METHOD FB_init : BOOL
VAR_INPUT
	bInitRetains : BOOL; // if TRUE, the retain variables are initialized (warm start / cold start)
	bInCopyCode : BOOL;  // if TRUE, the instance afterwards gets moved into the copy code (online change)
END_VAR
eObjectType := E_BACnetObjType.ObjAnalogValue;
END_METHOD

END_FUNCTION_BLOCK

// POUs/Remote/Objects/Basic/[Base]/FB_BACnetRM_EventObject
FUNCTION_BLOCK FB_BACnetRM_EventObject EXTENDS FB_BACnetRM_Object
VAR_OUTPUT
	bEvent						: BOOL;												// Indicates an active event
END_VAR
VAR
	{region 'Event'}
		stStatusFlags			: ST_BA_StatusFlags;
	{endregion}
END_VAR

SUPER^();

bEvent := F_BA_IsDisturbed(stStatusFlags);

METHOD PROTECTED OnObjectStateChanged
SUPER^.OnObjectStateChanged();

SyncProperty(E_BACnetPropIdentifier.PropStatusFlags, SIZEOF(stStatusFlags), ADR(stStatusFlags), E_BA_SyncModeRM.eRead);
END_METHOD

PROPERTY StatusFlags : ST_BA_StatusFlags
GET
StatusFlags := stStatusFlags;
END_GET
END_PROPERTY

END_FUNCTION_BLOCK

// POUs/Remote/Objects/Basic/FB_BACnetRM_AV_Disp
{attribute 'enable_dynamic_creation'}
FUNCTION_BLOCK FB_BACnetRM_AV_Disp EXTENDS FB_BACnetRM_Object
VAR_INPUT CONSTANT PERSISTENT
	{region 'Fixed Parameters'}
		{attribute 'parameterCategory':='Config'}
		fReadIncrement : REAL;
	{endregion}
END_VAR
VAR_OUTPUT
	fPresVal 	: REAL;
END_VAR

SUPER^();

METHOD PROTECTED OnObjectStateChanged
SUPER^.OnObjectStateChanged();

SyncPropertyReal(E_BACnetPropIdentifier.PropPresentValue, SIZEOF(fPresVal), ADR(fPresVal), E_BA_SyncModeRM.eRead, fReadIncrement);
END_METHOD

METHOD FB_init : BOOL
VAR_INPUT
	bInitRetains : BOOL; // if TRUE, the retain variables are initialized (warm start / cold start)
	bInCopyCode : BOOL;  // if TRUE, the instance afterwards gets moved into the copy code (online change)
END_VAR
eObjectType := E_BACnetObjType.ObjAnalogValue;
END_METHOD

END_FUNCTION_BLOCK

// POUs/Remote/Objects/Basic/FB_BACnetRM_AV_Setp
{attribute 'enable_dynamic_creation'}
FUNCTION_BLOCK FB_BACnetRM_AV_Setp EXTENDS FB_BACnetRM_Object
VAR_INPUT CONSTANT PERSISTENT
	{region 'Fixed Parameters'}
		{attribute 'parameterCategory':='Config'}
		fReadIncrement : REAL; 
		{attribute 'parameterCategory':='Config'}
		fWriteIncrement : REAL; 
	{endregion}
END_VAR
VAR_INPUT CONSTANT
	{region 'Operational Parameters'}
		{attribute 'parameterCategory':='Value'}
		fValue : REAL;
	{endregion}
END_VAR
VAR_OUTPUT
	fPresVal 	: REAL;
END_VAR

SUPER^();

{attribute 'hide'}
METHOD OnCOV
VAR_INPUT
	ePropID		: E_BACnetPropIdentifier;
END_VAR
CASE (ePropID) OF
	E_BACnetPropIdentifier.PropPresentValue:
		fValue := fPresVal;
		
ELSE
	SUPER^.OnCOV(ePropID);
END_CASE
END_METHOD

METHOD PROTECTED OnObjectStateChanged
SUPER^.OnObjectStateChanged();

SyncPropertyReal(E_BACnetPropIdentifier.PropPresentValue, SIZEOF(fPresVal), ADR(fPresVal), E_BA_SyncModeRM.eRead, fReadIncrement);

SyncPropertyReal(E_BACnetPropIdentifier.PropPresentValue, SIZEOF(fValue), ADR(fValue), E_BA_SyncModeRM.eWrite, fWriteIncrement);
END_METHOD

METHOD FB_init : BOOL
VAR_INPUT
	bInitRetains : BOOL; // if TRUE, the retain variables are initialized (warm start / cold start)
	bInCopyCode : BOOL;  // if TRUE, the instance afterwards gets moved into the copy code (online change)
END_VAR
eObjectType := E_BACnetObjType.ObjAnalogValue;
END_METHOD

END_FUNCTION_BLOCK

// POUs/Remote/Objects/Basic/FB_BACnetRM_AI
{attribute 'enable_dynamic_creation'}
FUNCTION_BLOCK FB_BACnetRM_AI EXTENDS FB_BACnetRM_EventObject
VAR_INPUT CONSTANT PERSISTENT
	{region 'Fixed Parameters'}
		{attribute 'parameterCategory':='Config'}
		fReadIncrement : REAL; 
	{endregion}
END_VAR
VAR_OUTPUT
	fPresVal 	: REAL;
END_VAR

SUPER^();

METHOD PROTECTED OnObjectStateChanged
SUPER^.OnObjectStateChanged();

SyncPropertyReal(E_BACnetPropIdentifier.PropPresentValue, SIZEOF(fPresVal), ADR(fPresVal), E_BA_SyncModeRM.eRead, fReadIncrement);
END_METHOD

METHOD FB_init : BOOL
VAR_INPUT
	bInitRetains : BOOL; // if TRUE, the retain variables are initialized (warm start / cold start)
	bInCopyCode : BOOL;  // if TRUE, the instance afterwards gets moved into the copy code (online change)
END_VAR
eObjectType := E_BACnetObjType.ObjAnalogInput;
END_METHOD

END_FUNCTION_BLOCK

// POUs/Remote/Objects/Basic/FB_BACnetRM_AO
{attribute 'enable_dynamic_creation'}
FUNCTION_BLOCK FB_BACnetRM_AO EXTENDS FB_BACnetRM_EventObject
VAR_INPUT
	bEnWrite	 	: BOOL;
	fVal 			: REAL;
	bNullVal 		: BOOL;
END_VAR
VAR_INPUT CONSTANT PERSISTENT
	{region 'Fixed Parameters'}
		{attribute 'parameterCategory':='Config'}
		fReadIncrement : REAL; 
		{attribute 'parameterCategory':='Config'}
		fWriteIncrement : REAL; 
			 
		{attribute 'parameterCategory':='Value'}
		ePriority : E_BACnet_Priority := BACnet_Param.eRemotePrio_Default;
	{endregion}
END_VAR
VAR_OUTPUT
	fPresVal 	: REAL;
END_VAR

SUPER^();

METHOD PROTECTED OnObjectStateChanged
SUPER^.OnObjectStateChanged();

SyncPropertyReal(E_BACnetPropIdentifier.PropPresentValue, SIZEOF(fPresVal), ADR(fPresVal), E_BA_SyncModeRM.eRead, fReadIncrement);

SyncPropertyPrioReal(E_BACnetPropIdentifier.PropPresentValue, SIZEOF(fVal), ADR(fVal), ADR(bEnWrite), ADR(bNullVal), ePriority, E_BA_SyncModeRM.eWrite, fWriteIncrement);
END_METHOD

METHOD FB_init : BOOL
VAR_INPUT
	bInitRetains : BOOL; // if TRUE, the retain variables are initialized (warm start / cold start)
	bInCopyCode : BOOL;  // if TRUE, the instance afterwards gets moved into the copy code (online change)
END_VAR
eObjectType := E_BACnetObjType.ObjAnalogOutput;
END_METHOD

END_FUNCTION_BLOCK

// POUs/Remote/Objects/Basic/FB_BACnetRM_BV
{attribute 'enable_dynamic_creation'}
FUNCTION_BLOCK FB_BACnetRM_BV EXTENDS FB_BACnetRM_EventObject
VAR_INPUT
	bEnWrite 		: BOOL;
	bVal 			: BOOL;
	bNullVal 		: BOOL;
END_VAR
VAR_INPUT CONSTANT PERSISTENT
	{region 'Fixed Parameters'}
		{attribute 'parameterCategory':='Value'}
		ePriority : E_BACnet_Priority := BACnet_Param.eRemotePrio_Default;
	{endregion}
END_VAR
VAR_OUTPUT
	bPresVal 	: BOOL;
END_VAR

SUPER^();

METHOD PROTECTED OnObjectStateChanged
SUPER^.OnObjectStateChanged();

SyncProperty(E_BACnetPropIdentifier.PropPresentValue, SIZEOF(bPresVal), ADR(bPresVal), E_BA_SyncModeRM.eRead);

SyncPropertyPrio(E_BACnetPropIdentifier.PropPresentValue, SIZEOF(bVal), ADR(bVal), ADR(bEnWrite), ADR(bNullVal), ePriority, E_BA_SyncModeRM.eWrite);
END_METHOD

METHOD FB_init : BOOL
VAR_INPUT
	bInitRetains : BOOL; // if TRUE, the retain variables are initialized (warm start / cold start)
	bInCopyCode : BOOL;  // if TRUE, the instance afterwards gets moved into the copy code (online change)
END_VAR
eObjectType := E_BACnetObjType.ObjBinaryValue;
END_METHOD

END_FUNCTION_BLOCK

// POUs/Remote/Objects/Basic/FB_BACnetRM_BV_Disp
{attribute 'enable_dynamic_creation'}
FUNCTION_BLOCK FB_BACnetRM_BV_Disp EXTENDS FB_BACnetRM_Object
VAR_OUTPUT
	bPresVal	: BOOL;
END_VAR

SUPER^();

METHOD PROTECTED OnObjectStateChanged
SUPER^.OnObjectStateChanged();

SyncProperty(E_BACnetPropIdentifier.PropPresentValue, SIZEOF(bPresVal), ADR(bPresVal), E_BA_SyncModeRM.eRead);
END_METHOD

METHOD FB_init : BOOL
VAR_INPUT
	bInitRetains : BOOL; // if TRUE, the retain variables are initialized (warm start / cold start)
	bInCopyCode : BOOL;  // if TRUE, the instance afterwards gets moved into the copy code (online change)
END_VAR
eObjectType := E_BACnetObjType.ObjBinaryValue;
END_METHOD

END_FUNCTION_BLOCK

// POUs/Remote/Objects/Basic/FB_BACnetRM_BV_Setp
{attribute 'enable_dynamic_creation'}
FUNCTION_BLOCK FB_BACnetRM_BV_Setp EXTENDS FB_BACnetRM_Object
VAR_INPUT CONSTANT
	{region 'Operational Parameters'}
		{attribute 'parameterCategory':='Value'}
		bValue : BOOL;
	{endregion}
END_VAR
VAR_OUTPUT
	bPresVal	: BOOL;
END_VAR

SUPER^();

{attribute 'hide'}
METHOD OnCOV
VAR_INPUT
	ePropID		: E_BACnetPropIdentifier;
END_VAR
CASE (ePropID) OF
	E_BACnetPropIdentifier.PropPresentValue:
		bValue := bPresVal;
		
ELSE
	SUPER^.OnCOV(ePropID);
END_CASE
END_METHOD

METHOD PROTECTED OnObjectStateChanged
SUPER^.OnObjectStateChanged();

SyncProperty(E_BACnetPropIdentifier.PropPresentValue, SIZEOF(bPresVal), ADR(bPresVal), E_BA_SyncModeRM.eRead);

SyncProperty(E_BACnetPropIdentifier.PropPresentValue, SIZEOF(bValue), ADR(bValue), E_BA_SyncModeRM.eWrite);
END_METHOD

METHOD FB_init : BOOL
VAR_INPUT
	bInitRetains : BOOL; // if TRUE, the retain variables are initialized (warm start / cold start)
	bInCopyCode : BOOL;  // if TRUE, the instance afterwards gets moved into the copy code (online change)
END_VAR
eObjectType := E_BACnetObjType.ObjBinaryValue;
END_METHOD

END_FUNCTION_BLOCK

// POUs/Remote/Objects/Basic/FB_BACnetRM_BI
{attribute 'enable_dynamic_creation'}
FUNCTION_BLOCK FB_BACnetRM_BI EXTENDS FB_BACnetRM_EventObject
VAR_OUTPUT
	bPresVal 	: BOOL;
END_VAR

SUPER^();

METHOD PROTECTED OnObjectStateChanged
SUPER^.OnObjectStateChanged();

SyncProperty(E_BACnetPropIdentifier.PropPresentValue, SIZEOF(bPresVal), ADR(bPresVal), E_BA_SyncModeRM.eRead);
END_METHOD

METHOD FB_init : BOOL
VAR_INPUT
	bInitRetains : BOOL; // if TRUE, the retain variables are initialized (warm start / cold start)
	bInCopyCode : BOOL;  // if TRUE, the instance afterwards gets moved into the copy code (online change)
END_VAR
eObjectType := E_BACnetObjType.ObjBinaryInput;
END_METHOD

END_FUNCTION_BLOCK

// POUs/Remote/Objects/Basic/FB_BACnetRM_BO
{attribute 'enable_dynamic_creation'}
FUNCTION_BLOCK FB_BACnetRM_BO EXTENDS FB_BACnetRM_EventObject
VAR_INPUT
	bEnWrite 		: BOOL;
	bVal 			: BOOL;
	bNullVal 		: BOOL;	
END_VAR
VAR_INPUT CONSTANT PERSISTENT
	{region 'Fixed Parameters'}
		{attribute 'parameterCategory':='Value'}
		ePriority : E_BACnet_Priority := BACnet_Param.eRemotePrio_Default;
	{endregion}
END_VAR
VAR_OUTPUT
	bPresVal 	: BOOL;
END_VAR

SUPER^();

METHOD PROTECTED OnObjectStateChanged
SUPER^.OnObjectStateChanged();

SyncProperty(E_BACnetPropIdentifier.PropPresentValue, SIZEOF(bPresVal), ADR(bPresVal), E_BA_SyncModeRM.eRead);

SyncPropertyPrio(E_BACnetPropIdentifier.PropPresentValue, SIZEOF(bVal), ADR(bVal), ADR(bEnWrite), ADR(bNullVal), ePriority, E_BA_SyncModeRM.eWrite);
END_METHOD

METHOD FB_init : BOOL
VAR_INPUT
	bInitRetains : BOOL; // if TRUE, the retain variables are initialized (warm start / cold start)
	bInCopyCode : BOOL;  // if TRUE, the instance afterwards gets moved into the copy code (online change)
END_VAR
eObjectType := E_BACnetObjType.ObjBinaryOutput;
END_METHOD

END_FUNCTION_BLOCK

// POUs/Remote/Objects/Basic/FB_BACnetRM_MV
{attribute 'enable_dynamic_creation'}
FUNCTION_BLOCK FB_BACnetRM_MV EXTENDS FB_BACnetRM_EventObject
VAR_INPUT
	bEnWrite 		: BOOL;
	nVal 			: UDINT;
	bNullVal 		: BOOL;	
END_VAR
VAR_INPUT CONSTANT PERSISTENT
	{region 'Fixed Parameters'}
		{attribute 'parameterCategory':='Value'}
		ePriority : E_BACnet_Priority := BACnet_Param.eRemotePrio_Default;
	{endregion}
END_VAR
VAR_OUTPUT
	nPresVal 	: UDINT;
END_VAR

SUPER^();

METHOD PROTECTED OnObjectStateChanged
SUPER^.OnObjectStateChanged();

SyncProperty(E_BACnetPropIdentifier.PropPresentValue, SIZEOF(nPresVal), ADR(nPresVal), E_BA_SyncModeRM.eRead);

SyncPropertyPrio(E_BACnetPropIdentifier.PropPresentValue, SIZEOF(nVal), ADR(nVal), ADR(bEnWrite), ADR(bNullVal), ePriority, E_BA_SyncModeRM.eWrite);
END_METHOD

METHOD FB_init : BOOL
VAR_INPUT
	bInitRetains : BOOL; // if TRUE, the retain variables are initialized (warm start / cold start)
	bInCopyCode : BOOL;  // if TRUE, the instance afterwards gets moved into the copy code (online change)
END_VAR
eObjectType := E_BACnetObjType.ObjMultistateValue;
END_METHOD

END_FUNCTION_BLOCK

// POUs/Remote/Objects/Basic/FB_BACnetRM_MV_Disp
{attribute 'enable_dynamic_creation'}
FUNCTION_BLOCK FB_BACnetRM_MV_Disp EXTENDS FB_BACnetRM_Object
VAR_OUTPUT
	nPresVal		: UDINT		:= 1;
END_VAR

SUPER^();

METHOD PROTECTED OnObjectStateChanged
SUPER^.OnObjectStateChanged();

SyncProperty(E_BACnetPropIdentifier.PropPresentValue, SIZEOF(nPresVal), ADR(nPresVal), E_BA_SyncModeRM.eRead);
END_METHOD

METHOD FB_init : BOOL
VAR_INPUT
	bInitRetains : BOOL; // if TRUE, the retain variables are initialized (warm start / cold start)
	bInCopyCode : BOOL;  // if TRUE, the instance afterwards gets moved into the copy code (online change)
END_VAR
eObjectType := E_BACnetObjType.ObjMultistateValue;
END_METHOD

END_FUNCTION_BLOCK

// POUs/Remote/Objects/Basic/FB_BACnetRM_MV_Setp
{attribute 'enable_dynamic_creation'}
FUNCTION_BLOCK FB_BACnetRM_MV_Setp EXTENDS FB_BACnetRM_Object
VAR_INPUT CONSTANT
	{region 'Operational Parameters'}
		{attribute 'parameterCategory':='Value'}
		nValue : UDINT;
	{endregion}
END_VAR
VAR_OUTPUT
	nPresVal		: UDINT		:= 1;
END_VAR

SUPER^();

{attribute 'hide'}
METHOD OnCOV
VAR_INPUT
	ePropID		: E_BACnetPropIdentifier;
END_VAR
CASE (ePropID) OF
	E_BACnetPropIdentifier.PropPresentValue:
		nValue := nPresVal;
		
ELSE
	SUPER^.OnCOV(ePropID);
END_CASE
END_METHOD

METHOD PROTECTED OnObjectStateChanged
SUPER^.OnObjectStateChanged();

SyncProperty(E_BACnetPropIdentifier.PropPresentValue, SIZEOF(nPresVal), ADR(nPresVal), E_BA_SyncModeRM.eRead);

SyncProperty(E_BACnetPropIdentifier.PropPresentValue, SIZEOF(nValue), ADR(nValue), E_BA_SyncModeRM.eWrite);
END_METHOD

METHOD FB_init : BOOL
VAR_INPUT
	bInitRetains : BOOL; // if TRUE, the retain variables are initialized (warm start / cold start)
	bInCopyCode : BOOL;  // if TRUE, the instance afterwards gets moved into the copy code (online change)
END_VAR
eObjectType := E_BACnetObjType.ObjMultistateValue;
END_METHOD

END_FUNCTION_BLOCK

// POUs/Remote/Objects/Basic/FB_BACnetRM_MI
{attribute 'enable_dynamic_creation'}
FUNCTION_BLOCK FB_BACnetRM_MI EXTENDS FB_BACnetRM_EventObject
VAR_OUTPUT
	nPresVal 	: UDINT;
END_VAR

SUPER^();

METHOD PROTECTED OnObjectStateChanged
SUPER^.OnObjectStateChanged();

SyncProperty(E_BACnetPropIdentifier.PropPresentValue, SIZEOF(nPresVal), ADR(nPresVal), E_BA_SyncModeRM.eRead);
END_METHOD

METHOD FB_init : BOOL
VAR_INPUT
	bInitRetains : BOOL; // if TRUE, the retain variables are initialized (warm start / cold start)
	bInCopyCode : BOOL;  // if TRUE, the instance afterwards gets moved into the copy code (online change)
END_VAR
eObjectType := E_BACnetObjType.ObjMultistateInput;
END_METHOD

END_FUNCTION_BLOCK

// POUs/Remote/Objects/Basic/FB_BACnetRM_MO
{attribute 'enable_dynamic_creation'}
FUNCTION_BLOCK FB_BACnetRM_MO EXTENDS FB_BACnetRM_EventObject
VAR_INPUT
	bEnWrite 		: BOOL;
	nVal 			: UDINT;
	bNullVal 		: BOOL;
END_VAR
VAR_INPUT CONSTANT PERSISTENT
	{region 'Fixed Parameters'}
		{attribute 'parameterCategory':='Value'}
		ePriority : E_BACnet_Priority := BACnet_Param.eRemotePrio_Default;
	{endregion}
END_VAR
VAR_OUTPUT
	nPresVal 	: UDINT;
END_VAR

SUPER^();

METHOD PROTECTED OnObjectStateChanged
SUPER^.OnObjectStateChanged();

SyncProperty(E_BACnetPropIdentifier.PropPresentValue, SIZEOF(nPresVal), ADR(nPresVal), E_BA_SyncModeRM.eRead);

SyncPropertyPrio(E_BACnetPropIdentifier.PropPresentValue, SIZEOF(nVal), ADR(nVal), ADR(bEnWrite), ADR(bNullVal), ePriority, E_BA_SyncModeRM.eWrite);
END_METHOD

METHOD FB_init : BOOL
VAR_INPUT
	bInitRetains : BOOL; // if TRUE, the retain variables are initialized (warm start / cold start)
	bInCopyCode : BOOL;  // if TRUE, the instance afterwards gets moved into the copy code (online change)
END_VAR
eObjectType := E_BACnetObjType.ObjMultistateOutput;
END_METHOD

END_FUNCTION_BLOCK

// POUs/Remote/Objects/Basic/FB_BACnetRM_TLog
{attribute 'enable_dynamic_creation'}
FUNCTION_BLOCK FB_BACnetRM_TLog EXTENDS FB_BACnetRM_BaseTLog
VAR_OUTPUT
	nRecCnt 	: UDINT;
	nTotRecCnt	: UDINT;
END_VAR

SUPER^();

METHOD PROTECTED OnObjectStateChanged
SUPER^.OnObjectStateChanged();

SyncProperty(E_BACnetPropIdentifier.PropRecordCount, SIZEOF(nRecCnt), ADR(nRecCnt), E_BA_SyncModeRM.eRead);
SyncProperty(E_BACnetPropIdentifier.PropTotalRecordCount, SIZEOF(nTotRecCnt), ADR(nTotRecCnt), E_BA_SyncModeRM.eRead);
END_METHOD

METHOD FB_init : BOOL
VAR_INPUT
	bInitRetains : BOOL; // if TRUE, the retain variables are initialized (warm start / cold start)
	bInCopyCode : BOOL;  // if TRUE, the instance afterwards gets moved into the copy code (online change)
END_VAR
eObjectType := E_BACnetObjType.ObjTrendLog;
END_METHOD

END_FUNCTION_BLOCK

// POUs/Remote/Objects/Basic/[Base]/FB_BACnetRM_BaseTLog
FUNCTION_BLOCK FB_BACnetRM_BaseTLog EXTENDS FB_BACnetRM_EventObject
VAR_OUTPUT
	nRecordCount				: UDINT;
	nTotalRecordCount			: UDINT;
END_VAR

SUPER^();

METHOD PROTECTED OnObjectStateChanged
SUPER^.OnObjectStateChanged();

SyncProperty(E_BACnetPropIdentifier.PropRecordCount, SIZEOF(nRecordCount), ADR(nRecordCount), E_BA_SyncModeRM.eRead);
SyncProperty(E_BACnetPropIdentifier.PropTotalRecordCount, SIZEOF(nTotalRecordCount), ADR(nTotalRecordCount), E_BA_SyncModeRM.eRead);
END_METHOD

END_FUNCTION_BLOCK

// POUs/Remote/Objects/Basic/FB_BACnetRM_TLM
{attribute 'enable_dynamic_creation'}
FUNCTION_BLOCK FB_BACnetRM_TLM EXTENDS FB_BACnetRM_BaseTLog
VAR_OUTPUT
	nRecCnt 	: UDINT;
	nTotRecCnt	: UDINT;
END_VAR

SUPER^();

METHOD PROTECTED OnObjectStateChanged
SUPER^.OnObjectStateChanged();

SyncProperty(E_BACnetPropIdentifier.PropRecordCount, SIZEOF(nRecCnt), ADR(nRecCnt), E_BA_SyncModeRM.eRead);
SyncProperty(E_BACnetPropIdentifier.PropTotalRecordCount, SIZEOF(nTotRecCnt), ADR(nTotRecCnt), E_BA_SyncModeRM.eRead);
END_METHOD

METHOD FB_init : BOOL
VAR_INPUT
	bInitRetains : BOOL; // if TRUE, the retain variables are initialized (warm start / cold start)
	bInCopyCode : BOOL;  // if TRUE, the instance afterwards gets moved into the copy code (online change)
END_VAR
eObjectType := E_BACnetObjType.ObjTrendLogMultiple;
END_METHOD

END_FUNCTION_BLOCK

// POUs/Remote/Objects/Basic/FB_BACnetRM_Cal
{attribute 'enable_dynamic_creation'}
FUNCTION_BLOCK FB_BACnetRM_Cal EXTENDS FB_BACnetRM_Object
VAR_OUTPUT
	bPresVal 	: BOOL;
END_VAR

SUPER^();

METHOD PROTECTED OnObjectStateChanged
SUPER^.OnObjectStateChanged();

SyncProperty(E_BACnetPropIdentifier.PropPresentValue, SIZEOF(bPresVal), ADR(bPresVal), E_BA_SyncModeRM.eRead);
END_METHOD

METHOD FB_init : BOOL
VAR_INPUT
	bInitRetains : BOOL; // if TRUE, the retain variables are initialized (warm start / cold start)
	bInCopyCode : BOOL;  // if TRUE, the instance afterwards gets moved into the copy code (online change)
END_VAR
eObjectType := E_BACnetObjType.ObjCalendar;
END_METHOD

END_FUNCTION_BLOCK

// POUs/Remote/Objects/Basic/FB_BACnetRM_SchedA
{attribute 'enable_dynamic_creation'}
FUNCTION_BLOCK FB_BACnetRM_SchedA EXTENDS FB_BACnetRM_Object
VAR_OUTPUT
	fPresVal 	: REAL;
END_VAR

SUPER^();

METHOD PROTECTED OnObjectStateChanged
SUPER^.OnObjectStateChanged();

SyncProperty(E_BACnetPropIdentifier.PropPresentValue, SIZEOF(fPresVal), ADR(fPresVal), E_BA_SyncModeRM.eRead);
END_METHOD

METHOD FB_init : BOOL
VAR_INPUT
	bInitRetains : BOOL; // if TRUE, the retain variables are initialized (warm start / cold start)
	bInCopyCode : BOOL;  // if TRUE, the instance afterwards gets moved into the copy code (online change)
END_VAR
eObjectType := E_BACnetObjType.ObjSchedule;
END_METHOD

END_FUNCTION_BLOCK

// POUs/Remote/Objects/Basic/FB_BACnetRM_SchedB
{attribute 'enable_dynamic_creation'}
FUNCTION_BLOCK FB_BACnetRM_SchedB EXTENDS FB_BACnetRM_Object
VAR_OUTPUT
	bPresVal 	: BOOL;
END_VAR

SUPER^();

METHOD PROTECTED OnObjectStateChanged
SUPER^.OnObjectStateChanged();

SyncProperty(E_BACnetPropIdentifier.PropPresentValue, SIZEOF(bPresVal), ADR(bPresVal), E_BA_SyncModeRM.eRead);
END_METHOD

METHOD FB_init : BOOL
VAR_INPUT
	bInitRetains : BOOL; // if TRUE, the retain variables are initialized (warm start / cold start)
	bInCopyCode : BOOL;  // if TRUE, the instance afterwards gets moved into the copy code (online change)
END_VAR
eObjectType := E_BACnetObjType.ObjSchedule;
END_METHOD

END_FUNCTION_BLOCK

// POUs/Remote/Objects/Basic/FB_BACnetRM_SchedM
{attribute 'enable_dynamic_creation'}
FUNCTION_BLOCK FB_BACnetRM_SchedM EXTENDS FB_BACnetRM_Object
VAR_OUTPUT
	nPresVal 	: UDINT;
END_VAR

SUPER^();

METHOD PROTECTED OnObjectStateChanged
SUPER^.OnObjectStateChanged();

SyncProperty(E_BACnetPropIdentifier.PropPresentValue, SIZEOF(nPresVal), ADR(nPresVal), E_BA_SyncModeRM.eRead);
END_METHOD

METHOD FB_init : BOOL
VAR_INPUT
	bInitRetains : BOOL; // if TRUE, the retain variables are initialized (warm start / cold start)
	bInCopyCode : BOOL;  // if TRUE, the instance afterwards gets moved into the copy code (online change)
END_VAR
eObjectType := E_BACnetObjType.ObjSchedule;
END_METHOD

END_FUNCTION_BLOCK

// POUs/Remote/Objects/Basic/FB_BACnetRM_Loop
{attribute 'enable_dynamic_creation'}
FUNCTION_BLOCK FB_BACnetRM_Loop EXTENDS FB_BACnetRM_EventObject
VAR_OUTPUT
	fPresVal			: REAL;
	fSetpoint			: REAL;
	fCtrlVar			: REAL;
END_VAR

SUPER^();

METHOD PROTECTED OnObjectStateChanged
SUPER^.OnObjectStateChanged();

SyncProperty(E_BACnetPropIdentifier.PropPresentValue, SIZEOF(fPresVal), ADR(fPresVal), E_BA_SyncModeRM.eRead);
SyncProperty(E_BACnetPropIdentifier.PropSetpoint, SIZEOF(fSetpoint), ADR(fSetpoint), E_BA_SyncModeRM.eRead);
SyncProperty(E_BACnetPropIdentifier.PropControlledVariableValue, SIZEOF(fCtrlVar), ADR(fCtrlVar), E_BA_SyncModeRM.eRead);
END_METHOD

METHOD FB_init : BOOL
VAR_INPUT
	bInitRetains : BOOL; // if TRUE, the retain variables are initialized (warm start / cold start)
	bInCopyCode : BOOL;  // if TRUE, the instance afterwards gets moved into the copy code (online change)
END_VAR
eObjectType := E_BACnetObjType.ObjLoop;
END_METHOD

END_FUNCTION_BLOCK

// POUs/Remote/Objects/Convenience/FB_BACnetRM_CnvLoop
{attribute 'enable_dynamic_creation'}
FUNCTION_BLOCK FB_BACnetRM_CnvLoop EXTENDS FB_BACnetRM_Loop
VAR_INPUT CONSTANT PERSISTENT
	{region 'Variable Parameters'}
		{attribute 'parameterCategory':='Config'}
		fProportionalConstant : REAL;
		{attribute 'parameterCategory':='Config'}
		eProportionalConstantUnit : E_BA_Unit;
		{attribute 'parameterCategory':='Config'}
		fIntegralConstant : REAL;
		{attribute 'parameterCategory':='Config'}
		eIntegralConstantUnit : E_BA_Unit;
		{attribute 'parameterCategory':='Config'}
		fDerivativeConstant : REAL;
		{attribute 'parameterCategory':='Config'}
		eDerivativeConstantUnit : E_BA_Unit;
	{endregion}
END_VAR

SUPER^();

METHOD PROTECTED OnObjectStateChanged
SUPER^.OnObjectStateChanged();

SyncProperty(E_BACnetPropIdentifier.PropProportionalConstant, SIZEOF(fProportionalConstant), ADR(fProportionalConstant), E_BA_SyncModeRM.eRead);
SyncProperty(E_BACnetPropIdentifier.PropProportionalConstantUnits, SIZEOF(eProportionalConstantUnit), ADR(eProportionalConstantUnit), E_BA_SyncModeRM.eRead);
SyncProperty(E_BACnetPropIdentifier.PropIntegralConstant, SIZEOF(fIntegralConstant), ADR(fIntegralConstant), E_BA_SyncModeRM.eRead);
SyncProperty(E_BACnetPropIdentifier.PropIntegralConstantUnits, SIZEOF(eIntegralConstantUnit), ADR(eIntegralConstantUnit), E_BA_SyncModeRM.eRead);
SyncProperty(E_BACnetPropIdentifier.PropDerivativeConstant, SIZEOF(fDerivativeConstant), ADR(fDerivativeConstant), E_BA_SyncModeRM.eRead);
SyncProperty(E_BACnetPropIdentifier.PropDerivativeConstantUnits, SIZEOF(eDerivativeConstantUnit), ADR(eDerivativeConstantUnit), E_BA_SyncModeRM.eRead);
END_METHOD

END_FUNCTION_BLOCK

// POUs/Remote/Objects/Basic/FB_BACnetRM_File
{attribute 'enable_dynamic_creation'}
FUNCTION_BLOCK FB_BACnetRM_File EXTENDS FB_BACnetRM_Object
VAR_OUTPUT
	nFileSize		: UDINT;
END_VAR

SUPER^();

METHOD PROTECTED OnObjectStateChanged
SUPER^.OnObjectStateChanged();

SyncProperty(E_BACnetPropIdentifier.PropFileSize, SIZEOF(nFileSize), ADR(nFileSize), E_BA_SyncModeRM.eRead);
END_METHOD

METHOD FB_init : BOOL
VAR_INPUT
	bInitRetains : BOOL; // if TRUE, the retain variables are initialized (warm start / cold start)
	bInCopyCode : BOOL;  // if TRUE, the instance afterwards gets moved into the copy code (online change)
END_VAR
eObjectType := E_BACnetObjType.ObjFile;
END_METHOD

END_FUNCTION_BLOCK

// POUs/Remote/Objects/Basic/FB_BACnetRM_NC
{attribute 'enable_dynamic_creation'}
FUNCTION_BLOCK FB_BACnetRM_NC EXTENDS FB_BACnetRM_Object

SUPER^();

METHOD FB_init : BOOL
VAR_INPUT
	bInitRetains : BOOL; // if TRUE, the retain variables are initialized (warm start / cold start)
	bInCopyCode : BOOL;  // if TRUE, the instance afterwards gets moved into the copy code (online change)
END_VAR
eObjectType := E_BACnetObjType.ObjNotificationClass;
END_METHOD

END_FUNCTION_BLOCK

// POUs/Remote/Objects/Basic/FB_BACnetRM_Acc
{attribute 'enable_dynamic_creation'}
FUNCTION_BLOCK FB_BACnetRM_Acc EXTENDS FB_BACnetRM_EventObject
VAR_OUTPUT
	nPresVal			: UDINT;
END_VAR

SUPER^();

METHOD PROTECTED OnObjectStateChanged
SUPER^.OnObjectStateChanged();

SyncProperty(E_BACnetPropIdentifier.PropPresentValue, SIZEOF(nPresVal), ADR(nPresVal), E_BA_SyncModeRM.eRead);
END_METHOD

METHOD FB_init : BOOL
VAR_INPUT
	bInitRetains : BOOL; // if TRUE, the retain variables are initialized (warm start / cold start)
	bInCopyCode : BOOL;  // if TRUE, the instance afterwards gets moved into the copy code (online change)
END_VAR
eObjectType := E_BACnetObjType.ObjAccumulator;
END_METHOD

END_FUNCTION_BLOCK

// POUs/Remote/Objects/Basic/FB_BACnetRM_PC
{attribute 'enable_dynamic_creation'}
FUNCTION_BLOCK FB_BACnetRM_PC EXTENDS FB_BACnetRM_EventObject
VAR_OUTPUT
	fPresVal			: REAL;
END_VAR

SUPER^();

METHOD PROTECTED OnObjectStateChanged
SUPER^.OnObjectStateChanged();

SyncProperty(E_BACnetPropIdentifier.PropPresentValue, SIZEOF(fPresVal), ADR(fPresVal), E_BA_SyncModeRM.eRead);
END_METHOD

METHOD FB_init : BOOL
VAR_INPUT
	bInitRetains : BOOL; // if TRUE, the retain variables are initialized (warm start / cold start)
	bInCopyCode : BOOL;  // if TRUE, the instance afterwards gets moved into the copy code (online change)
END_VAR
eObjectType := E_BACnetObjType.ObjPulseConverter;
END_METHOD

END_FUNCTION_BLOCK

// POUs/Remote/Objects/Basic/FB_BACnetRM_Prog
{attribute 'enable_dynamic_creation'}
FUNCTION_BLOCK FB_BACnetRM_Prog EXTENDS FB_BACnetRM_EventObject
VAR_OUTPUT
	eState			: E_BACnet_ProgramState;
END_VAR

SUPER^();

METHOD PROTECTED OnObjectStateChanged
SUPER^.OnObjectStateChanged();

SyncProperty(E_BACnetPropIdentifier.PropProgramState, SIZEOF(eState), ADR(eState), E_BA_SyncModeRM.eRead);
END_METHOD

METHOD FB_init : BOOL
VAR_INPUT
	bInitRetains : BOOL; // if TRUE, the retain variables are initialized (warm start / cold start)
	bInCopyCode : BOOL;  // if TRUE, the instance afterwards gets moved into the copy code (online change)
END_VAR
eObjectType := E_BACnetObjType.ObjProg;
END_METHOD

END_FUNCTION_BLOCK

// POUs/Remote/Objects/Basic/FB_BACnetRM_Avg
{attribute 'enable_dynamic_creation'}
FUNCTION_BLOCK FB_BACnetRM_Avg EXTENDS FB_BACnetRM_Object
VAR_OUTPUT
	fAvgVal			: REAL;
	fMinVal			: REAL;
	fMaxVal			: REAL;
END_VAR

SUPER^();

METHOD PROTECTED OnObjectStateChanged
VAR
	nPresentValue: INT;
END_VAR
SUPER^.OnObjectStateChanged();

SyncProperty(E_BACnetPropIdentifier.PropAverageValue, SIZEOF(fAvgVal), ADR(fAvgVal), E_BA_SyncModeRM.eRead);
SyncProperty(E_BACnetPropIdentifier.PropMinimumValue, SIZEOF(fMinVal), ADR(fMinVal), E_BA_SyncModeRM.eRead);
SyncProperty(E_BACnetPropIdentifier.PropMaximumValue, SIZEOF(fMaxVal), ADR(fMaxVal), E_BA_SyncModeRM.eRead);
END_METHOD

METHOD FB_init : BOOL
VAR_INPUT
	bInitRetains : BOOL; // if TRUE, the retain variables are initialized (warm start / cold start)
	bInCopyCode : BOOL;  // if TRUE, the instance afterwards gets moved into the copy code (online change)
END_VAR
eObjectType := E_BACnetObjType.ObjAveraging;
END_METHOD

END_FUNCTION_BLOCK

// POUs/Remote/Objects/Basic/FB_BACnetRM_Cmd
{attribute 'enable_dynamic_creation'}
FUNCTION_BLOCK FB_BACnetRM_Cmd EXTENDS FB_BACnetRM_Object
VAR_OUTPUT
	nPresVal			: UDINT;
	bAllWritesOk		: BOOL; (* all actions in selected action list are written *)
	bInProcess			: BOOL; (* object is busy *)
END_VAR

SUPER^();

METHOD PROTECTED OnObjectStateChanged
SUPER^.OnObjectStateChanged();

SyncProperty(E_BACnetPropIdentifier.PropPresentValue, SIZEOF(nPresVal), ADR(nPresVal), E_BA_SyncModeRM.eRead);
SyncProperty(E_BACnetPropIdentifier.PropAllWritesSuccessful, SIZEOF(bAllWritesOk), ADR(bAllWritesOk), E_BA_SyncModeRM.eRead);
SyncProperty(E_BACnetPropIdentifier.PropInProcess, SIZEOF(bInProcess), ADR(bInProcess), E_BA_SyncModeRM.eRead);
END_METHOD

METHOD FB_init : BOOL
VAR_INPUT
	bInitRetains : BOOL; // if TRUE, the retain variables are initialized (warm start / cold start)
	bInCopyCode : BOOL;  // if TRUE, the instance afterwards gets moved into the copy code (online change)
END_VAR
eObjectType := E_BACnetObjType.ObjCommand;
END_METHOD

END_FUNCTION_BLOCK

// POUs/Remote/Objects/Basic/FB_BACnetRM_Device
{attribute 'enable_dynamic_creation'}
FUNCTION_BLOCK FB_BACnetRM_Device EXTENDS FB_BACnetRM_Object
VAR_OUTPUT
	bOperational		: BOOL;
END_VAR

IF (NOT bReady) THEN
	IF (nObjectInstance = BACnet_Globals.nBACnetInstId_Auto) THEN
		nObjectInstance:=Client.ObjectInstance;
	END_IF
END_IF

SUPER^();

METHOD PROTECTED OnObjectStateChanged
SUPER^.OnObjectStateChanged();

IF (nObjectInstance = 16#23FFFFF) THEN
	nObjectInstance := Client.ObjectInstance;
END_IF

SyncProperty(E_BACnetPropIdentifier.PropSystemStatus, SIZEOF(bOperational), ADR(bOperational), E_BA_SyncModeRM.eRead);
END_METHOD

METHOD FB_init : BOOL
VAR_INPUT
	bInitRetains : BOOL; // if TRUE, the retain variables are initialized (warm start / cold start)
	bInCopyCode : BOOL;  // if TRUE, the instance afterwards gets moved into the copy code (online change)
END_VAR
eObjectType := E_BACnetObjType.ObjDevice;
END_METHOD

END_FUNCTION_BLOCK

// POUs/Remote/Objects/Basic/FB_BACnetRM_EE
{attribute 'enable_dynamic_creation'}
FUNCTION_BLOCK FB_BACnetRM_EE EXTENDS FB_BACnetRM_Object
VAR_OUTPUT
END_VAR

SUPER^();

METHOD PROTECTED OnObjectStateChanged
SUPER^.OnObjectStateChanged();
END_METHOD

METHOD FB_init : BOOL
VAR_INPUT
	bInitRetains : BOOL; // if TRUE, the retain variables are initialized (warm start / cold start)
	bInCopyCode : BOOL;  // if TRUE, the instance afterwards gets moved into the copy code (online change)
END_VAR
eObjectType := E_BACnetObjType.ObjEventEnrollment;
END_METHOD

END_FUNCTION_BLOCK

// POUs/Remote/Objects/Basic/FB_BACnetRM_ELog
{attribute 'enable_dynamic_creation'}
FUNCTION_BLOCK FB_BACnetRM_ELog EXTENDS FB_BACnetRM_BaseTLog

SUPER^();

METHOD FB_init : BOOL
VAR_INPUT
	bInitRetains : BOOL; // if TRUE, the retain variables are initialized (warm start / cold start)
	bInCopyCode : BOOL;  // if TRUE, the instance afterwards gets moved into the copy code (online change)
END_VAR
eObjectType := E_BACnetObjType.ObjEventLog;
END_METHOD

END_FUNCTION_BLOCK

// POUs/Remote/Objects/Basic/FB_BACnetRM_Group
{attribute 'enable_dynamic_creation'}
FUNCTION_BLOCK FB_BACnetRM_Group EXTENDS FB_BACnetRM_Object

SUPER^();

METHOD PROTECTED OnObjectStateChanged
SUPER^.OnObjectStateChanged();
END_METHOD

METHOD FB_init : BOOL
VAR_INPUT
	bInitRetains : BOOL; // if TRUE, the retain variables are initialized (warm start / cold start)
	bInCopyCode : BOOL;  // if TRUE, the instance afterwards gets moved into the copy code (online change)
END_VAR
eObjectType := E_BACnetObjType.ObjGroup;
END_METHOD

END_FUNCTION_BLOCK

// POUs/Remote/Objects/Experimental/FB_BACnetRM_ExpAV01
{attribute 'enable_dynamic_creation'}
{attribute 'hide'}	// (BETA) ...FB is only for testing!
FUNCTION_BLOCK FB_BACnetRM_ExpAV01 EXTENDS FB_BACnetRM_AV
VAR
	{region 'Test Properties'}
//		bHighLimitEnable		: BOOL;
//		fHighLimit				: REAL;
//		bLowLimitEnable			: BOOL;
//		fLowLimit				: REAL;
			 
		bWriteEnable			: BOOL;
		stLimitEnable 			: ST_BACnet_LimitEnableBits;
		stEventEnable 			: ST_BACnet_EventTransitionBits;		  
					   
		eReliability			: E_BA_Reliability;
		stAckedTransitions		: ST_BA_EventTransitions;
		eEventState				: E_BACnet_EventState;
	{endregion}
END_VAR

SUPER^();

METHOD PROTECTED OnObjectStateChanged
SUPER^.OnObjectStateChanged();

SyncProperty(E_BACnetPropIdentifier.PropReliability, SIZEOF(eReliability), ADR(eReliability), E_BA_SyncModeRM.eRead);
SyncProperty(E_BACnetPropIdentifier.PropEventState, SIZEOF(eEventState), ADR(eEventState), E_BA_SyncModeRM.eRead);
SyncProperty(E_BACnetPropIdentifier.PropAckedTransitions, SIZEOF(stAckedTransitions), ADR(stAckedTransitions), E_BA_SyncModeRM.eRead);


SyncPropertyEnable(E_BACnetPropIdentifier.PropEventEnable, SIZEOF(stEventEnable), ADR(stEventEnable), ADR(bWriteEnable), E_BA_SyncModeRM.eWrite);
SyncPropertyEnable(E_BACnetPropIdentifier.PropLimitEnable, SIZEOF(stLimitEnable), ADR(stLimitEnable), ADR(bWriteEnable), E_BA_SyncModeRM.eWrite);
END_METHOD

END_FUNCTION_BLOCK

// POUs/Remote/Objects/Experimental/FB_BACnetRM_ExpAV02
{attribute 'enable_dynamic_creation'}
{attribute 'hide'}	// (BETA) ...FB is only for testing!
FUNCTION_BLOCK FB_BACnetRM_ExpAV02 EXTENDS FB_BACnetRM_AV
VAR
	{region 'Test Properties'}
		stLimitEnable 			: ST_BACnet_LimitEnableBits;
	{endregion}
END_VAR
VAR
	{attribute 'hide'}
	fbLmEnWrite					: FB_BACnetRM_WriteProperty		:= (pData:=ADR(stLimitEnable), nData:=SIZEOF(stLimitEnable), ePropID:=PropLimitEnable, iObject:=THIS^);
	{attribute 'hide'}
	fbLmEnTrig					: FB_BA_ATrigCOV;
END_VAR

SUPER^();

IF (Client.bReady) THEN
	fbLmEnTrig(xValue:=stLimitEnable);
	fbLmEnWrite(Client:=Client, bExecute:=fbLmEnTrig.bQ);
END_IF

END_FUNCTION_BLOCK

// POUs/Remote/Objects/Primitive/FB_BACnetRM_BitString
{attribute 'enable_dynamic_creation'}
FUNCTION_BLOCK FB_BACnetRM_BitString EXTENDS FB_BACnetRM_Object
VAR_OUTPUT
	nPresVal 	: ULINT;
END_VAR

SUPER^();

METHOD PROTECTED OnObjectStateChanged
SUPER^.OnObjectStateChanged();

SyncProperty(E_BACnetPropIdentifier.PropPresentValue, SIZEOF(nPresVal), ADR(nPresVal), E_BA_SyncModeRM.eRead);
END_METHOD

METHOD FB_init : BOOL
VAR_INPUT
	bInitRetains : BOOL; // if TRUE, the retain variables are initialized (warm start / cold start)
	bInCopyCode : BOOL;  // if TRUE, the instance afterwards gets moved into the copy code (online change)
END_VAR
eObjectType := E_BACnetObjType.ObjBitStringValue;
END_METHOD

END_FUNCTION_BLOCK

// POUs/Remote/Objects/Primitive/FB_BACnetRM_ByteArr
{attribute 'enable_dynamic_creation'}
FUNCTION_BLOCK FB_BACnetRM_ByteArr EXTENDS FB_BACnetRM_Object
VAR_OUTPUT
	aPresVal 		: ARRAY [0..255] OF BYTE;
	nPresVal 		: UINT;
END_VAR

SUPER^();

METHOD PROTECTED OnObjectStateChanged
SUPER^.OnObjectStateChanged();

SyncProperty(E_BACnetPropIdentifier.PropPresentValue, SIZEOF(aPresVal), ADR(aPresVal), E_BA_SyncModeRM.eRead);
END_METHOD

METHOD FB_init : BOOL
VAR_INPUT
	bInitRetains : BOOL; // if TRUE, the retain variables are initialized (warm start / cold start)
	bInCopyCode : BOOL;  // if TRUE, the instance afterwards gets moved into the copy code (online change)
END_VAR
eObjectType := E_BACnetObjType.ObjOctetStringValue;
END_METHOD

END_FUNCTION_BLOCK

// POUs/Remote/Objects/Primitive/FB_BACnetRM_Date
{attribute 'enable_dynamic_creation'}
FUNCTION_BLOCK FB_BACnetRM_Date EXTENDS FB_BACnetRM_Object
VAR_OUTPUT
	stPresVal 	: ST_BA_Date;
END_VAR

SUPER^();

METHOD PROTECTED OnObjectStateChanged
SUPER^.OnObjectStateChanged();

SyncProperty(E_BACnetPropIdentifier.PropPresentValue, SIZEOF(stPresVal), ADR(stPresVal), E_BA_SyncModeRM.eRead);
END_METHOD

METHOD FB_init : BOOL
VAR_INPUT
	bInitRetains : BOOL; // if TRUE, the retain variables are initialized (warm start / cold start)
	bInCopyCode : BOOL;  // if TRUE, the instance afterwards gets moved into the copy code (online change)
END_VAR
eObjectType := E_BACnetObjType.ObjDateValue;
END_METHOD

END_FUNCTION_BLOCK

// POUs/Remote/Objects/Primitive/FB_BACnetRM_DateP
{attribute 'enable_dynamic_creation'}
FUNCTION_BLOCK FB_BACnetRM_DateP EXTENDS FB_BACnetRM_Object
VAR_OUTPUT
	stPresVal 	: ST_BA_Date;
END_VAR

SUPER^();

METHOD PROTECTED OnObjectStateChanged
SUPER^.OnObjectStateChanged();

SyncProperty(E_BACnetPropIdentifier.PropPresentValue, SIZEOF(stPresVal), ADR(stPresVal), E_BA_SyncModeRM.eRead);
END_METHOD

METHOD FB_init : BOOL
VAR_INPUT
	bInitRetains : BOOL; // if TRUE, the retain variables are initialized (warm start / cold start)
	bInCopyCode : BOOL;  // if TRUE, the instance afterwards gets moved into the copy code (online change)
END_VAR
eObjectType := E_BACnetObjType.ObjDatePatternValue;
END_METHOD

END_FUNCTION_BLOCK

// POUs/Remote/Objects/Primitive/FB_BACnetRM_DateTime
{attribute 'enable_dynamic_creation'}
FUNCTION_BLOCK FB_BACnetRM_DateTime EXTENDS FB_BACnetRM_Object
VAR_OUTPUT
	stPresVal 	: ST_BA_DateTime;
END_VAR

SUPER^();

METHOD PROTECTED OnObjectStateChanged
SUPER^.OnObjectStateChanged();

SyncProperty(E_BACnetPropIdentifier.PropPresentValue, SIZEOF(stPresVal), ADR(stPresVal), E_BA_SyncModeRM.eRead);
END_METHOD

METHOD FB_init : BOOL
VAR_INPUT
	bInitRetains : BOOL; // if TRUE, the retain variables are initialized (warm start / cold start)
	bInCopyCode : BOOL;  // if TRUE, the instance afterwards gets moved into the copy code (online change)
END_VAR
eObjectType := E_BACnetObjType.ObjDateTimeValue;
END_METHOD

END_FUNCTION_BLOCK

// POUs/Remote/Objects/Primitive/FB_BACnetRM_DateTimeP
{attribute 'enable_dynamic_creation'}
FUNCTION_BLOCK FB_BACnetRM_DateTimeP EXTENDS FB_BACnetRM_Object
VAR_OUTPUT
	stPresVal 	: ST_BA_DateTime;
END_VAR

SUPER^();

METHOD PROTECTED OnObjectStateChanged
SUPER^.OnObjectStateChanged();

SyncProperty(E_BACnetPropIdentifier.PropPresentValue, SIZEOF(stPresVal), ADR(stPresVal), E_BA_SyncModeRM.eRead);
END_METHOD

METHOD FB_init : BOOL
VAR_INPUT
	bInitRetains : BOOL; // if TRUE, the retain variables are initialized (warm start / cold start)
	bInCopyCode : BOOL;  // if TRUE, the instance afterwards gets moved into the copy code (online change)
END_VAR
eObjectType := E_BACnetObjType.ObjDateTimePatternValue;
END_METHOD

END_FUNCTION_BLOCK

// POUs/Remote/Objects/Primitive/FB_BACnetRM_Int
{attribute 'enable_dynamic_creation'}
FUNCTION_BLOCK FB_BACnetRM_Int EXTENDS FB_BACnetRM_Object
VAR_OUTPUT
	nPresVal 	: DINT;
END_VAR

SUPER^();

METHOD PROTECTED OnObjectStateChanged
SUPER^.OnObjectStateChanged();

SyncProperty(E_BACnetPropIdentifier.PropPresentValue, SIZEOF(nPresVal), ADR(nPresVal), E_BA_SyncModeRM.eRead);
END_METHOD

METHOD FB_init : BOOL
VAR_INPUT
	bInitRetains : BOOL; // if TRUE, the retain variables are initialized (warm start / cold start)
	bInCopyCode : BOOL;  // if TRUE, the instance afterwards gets moved into the copy code (online change)
END_VAR
eObjectType := E_BACnetObjType.ObjIntegerValue;
END_METHOD

END_FUNCTION_BLOCK

// POUs/Remote/Objects/Primitive/FB_BACnetRM_LAV
{attribute 'enable_dynamic_creation'}
FUNCTION_BLOCK FB_BACnetRM_LAV EXTENDS FB_BACnetRM_Object
VAR_OUTPUT
	fPresVal 	: LREAL;
END_VAR

SUPER^();

METHOD PROTECTED OnObjectStateChanged
SUPER^.OnObjectStateChanged();

SyncProperty(E_BACnetPropIdentifier.PropPresentValue, SIZEOF(fPresVal), ADR(fPresVal), E_BA_SyncModeRM.eRead);
END_METHOD

METHOD FB_init : BOOL
VAR_INPUT
	bInitRetains : BOOL; // if TRUE, the retain variables are initialized (warm start / cold start)
	bInCopyCode : BOOL;  // if TRUE, the instance afterwards gets moved into the copy code (online change)
END_VAR
eObjectType := E_BACnetObjType.ObjLargeAnalogValue;
END_METHOD

END_FUNCTION_BLOCK

// POUs/Remote/Objects/Primitive/FB_BACnetRM_String
{attribute 'enable_dynamic_creation'}
FUNCTION_BLOCK FB_BACnetRM_String EXTENDS FB_BACnetRM_Object
VAR_OUTPUT
	sPresVal 	: STRING;
END_VAR

SUPER^();

METHOD PROTECTED OnObjectStateChanged
SUPER^.OnObjectStateChanged();

SyncProperty(E_BACnetPropIdentifier.PropPresentValue, SIZEOF(sPresVal), ADR(sPresVal), E_BA_SyncModeRM.eRead);
END_METHOD

METHOD FB_init : BOOL
VAR_INPUT
	bInitRetains : BOOL; // if TRUE, the retain variables are initialized (warm start / cold start)
	bInCopyCode : BOOL;  // if TRUE, the instance afterwards gets moved into the copy code (online change)
END_VAR
eObjectType := E_BACnetObjType.ObjCharacterStringValue;
END_METHOD

END_FUNCTION_BLOCK

// POUs/Remote/Objects/Primitive/FB_BACnetRM_Time
{attribute 'enable_dynamic_creation'}
FUNCTION_BLOCK FB_BACnetRM_Time EXTENDS FB_BACnetRM_Object
VAR_OUTPUT
	stPresVal 	: ST_BA_Time;
END_VAR

SUPER^();

METHOD PROTECTED OnObjectStateChanged
SUPER^.OnObjectStateChanged();

SyncProperty(E_BACnetPropIdentifier.PropPresentValue, SIZEOF(stPresVal), ADR(stPresVal), E_BA_SyncModeRM.eRead);
END_METHOD

METHOD FB_init : BOOL
VAR_INPUT
	bInitRetains : BOOL; // if TRUE, the retain variables are initialized (warm start / cold start)
	bInCopyCode : BOOL;  // if TRUE, the instance afterwards gets moved into the copy code (online change)
END_VAR
eObjectType := E_BACnetObjType.ObjTimeValue;
END_METHOD

END_FUNCTION_BLOCK

// POUs/Remote/Objects/Primitive/FB_BACnetRM_TimeP
{attribute 'enable_dynamic_creation'}
FUNCTION_BLOCK FB_BACnetRM_TimeP EXTENDS FB_BACnetRM_Object
VAR_OUTPUT
	stPresVal 	: ST_BA_Time;
END_VAR

SUPER^();

METHOD PROTECTED OnObjectStateChanged
SUPER^.OnObjectStateChanged();

SyncProperty(E_BACnetPropIdentifier.PropPresentValue, SIZEOF(stPresVal), ADR(stPresVal), E_BA_SyncModeRM.eRead);
END_METHOD

METHOD FB_init : BOOL
VAR_INPUT
	bInitRetains : BOOL; // if TRUE, the retain variables are initialized (warm start / cold start)
	bInCopyCode : BOOL;  // if TRUE, the instance afterwards gets moved into the copy code (online change)
END_VAR
eObjectType := E_BACnetObjType.ObjTimePatternValue;
END_METHOD

END_FUNCTION_BLOCK

// POUs/Remote/Objects/Primitive/FB_BACnetRM_UInt
{attribute 'enable_dynamic_creation'}
FUNCTION_BLOCK FB_BACnetRM_UInt EXTENDS FB_BACnetRM_Object
VAR_OUTPUT
	nPresVal 	: UDINT;
END_VAR

SUPER^();

METHOD PROTECTED OnObjectStateChanged
SUPER^.OnObjectStateChanged();

SyncProperty(E_BACnetPropIdentifier.PropPresentValue, SIZEOF(nPresVal), ADR(nPresVal), E_BA_SyncModeRM.eRead);
END_METHOD

METHOD FB_init : BOOL
VAR_INPUT
	bInitRetains : BOOL; // if TRUE, the retain variables are initialized (warm start / cold start)
	bInCopyCode : BOOL;  // if TRUE, the instance afterwards gets moved into the copy code (online change)
END_VAR
eObjectType := E_BACnetObjType.ObjPositiveIntegerValue;
END_METHOD

END_FUNCTION_BLOCK

// POUs/Remote/Properties/FB_BACnetRM_ReadPropertyEx
FUNCTION_BLOCK FB_BACnetRM_ReadPropertyEx EXTENDS FB_BACnetRM_ReadProperty
VAR_INPUT
	nObjInst 	: UDINT;
	eObjType	: E_BACnetObjType;
END_VAR
VAR_OUTPUT
END_VAR
VAR
	refObj : FB_BACnetRM_Object;
	bRefObjUsed : BOOL;
END_VAR

IF iObject = 0 THEN
	iObject := refObj;
	bRefObjUsed:=TRUE;
END_IF

IF bRefObjUsed THEN
	refObj.ObjectInstance:=nObjInst;
	refObj.ObjectType:=eObjType;
END_IF

SUPER^();

END_FUNCTION_BLOCK

// POUs/Remote/Properties/FB_BACnetRM_WritePropertyEx
FUNCTION_BLOCK FB_BACnetRM_WritePropertyEx EXTENDS FB_BACnetRM_WriteProperty
VAR_INPUT
	nObjInst 	: UDINT;
	eObjType	: E_BACnetObjType;
END_VAR
VAR_OUTPUT
END_VAR
VAR
	refObj : FB_BACnetRM_Object;
	bRefObjUsed : BOOL;
END_VAR

IF iObject = 0 THEN
	iObject := refObj;
	bRefObjUsed:=TRUE;
END_IF

IF bRefObjUsed THEN
	refObj.ObjectInstance:=nObjInst;
	refObj.ObjectType:=eObjType;
END_IF

SUPER^();

END_FUNCTION_BLOCK

// POUs/Remote/Requests/[Internal]/FB_BACnetRM_ReqAckAlarm
{attribute 'c++_compatible'}
{attribute 'enable_dynamic_creation'}
{attribute 'hide'}
FUNCTION_BLOCK FB_BACnetRM_ReqAckAlarm EXTENDS FB_BACnetRM_ReqBase IMPLEMENTS ITcIoBACnetServiceResponseSink
VAR_INPUT
	sMsg : STRING;
	eAckEvent : E_BACnet_EventState;
END_VAR
VAR_OUTPUT
	bTsReady : BOOL;
	bReady : BOOL;
END_VAR
VAR
	req : AcknowledgeAlarmRequest;
	readTsReq : FB_BACnetRM_ReqRead;
	eventTs : ST_BACnet_EventTimeStamps;
END_VAR

IF NOT bTsReady THEN
	bTsReady := readTsReq.bReady;
END_IF

{attribute 'c++_compatible'}
{attribute 'minimal_input_size' := '4'}
{attribute 'pack_mode' := '4'}
{attribute 'hide'}
METHOD OnSendPropertyDataRequest : HRESULT
VAR_INPUT
	pResult	: POINTER TO SendDataRequestResult;
END_VAR
IF (pResult <> 0) THEN
	IF F_BACnetRM_IsErrorSet(pResult) THEN
		bReady := FALSE;
		OnSendPropertyDataRequest:=S_FALSE;
	ELSE
		bReady := FALSE;	
	END_IF
END_IF
END_METHOD

{attribute 'hide'}
METHOD Send : BOOL
VAR
	_ClTmp : ITcIoBACnetPlcClient;
END_VAR
IF Valid THEN
	req.acknowledgingProcessIdentifier := 0;
	req.eventObjectIdentifier := iObject.ObjectID;
	req.acknowledgmentSource := sMsg;
	req.eventStateAcknowledged := eAckEvent;
	IF eAckEvent = E_BACnet_EventState.eNormal THEN
		MEMCPY(ADR(req.timeStamp),ADR(eventTs.stToNormal), SIZEOF(ST_BACnet_TimeStampDateTime));
	ELSIF eAckEvent = E_BACnet_EventState.eFault THEN
		MEMCPY(ADR(req.timeStamp),ADR(eventTs.stToFault), SIZEOF(ST_BACnet_TimeStampDateTime));
	ELSE
		MEMCPY(ADR(req.timeStamp),ADR(eventTs.stToOffNormal), SIZEOF(ST_BACnet_TimeStampDateTime));
	END_IF
	
	_ClTmp := Client.iClient;
	
	IF S_OK = _ClTmp.AcknowledgeAlarm(ADR(req), Client.ObjectInstance, THIS^) THEN
		Send:=TRUE;
	END_IF
END_IF
END_METHOD

{attribute 'c++_compatible'}
{attribute 'minimal_input_size' := '4'}
{attribute 'pack_mode' := '4'}
{attribute 'hide'}
METHOD TcAddRef : UDINT
END_METHOD

{attribute 'c++_compatible'}
{attribute 'minimal_input_size' := '4'}
{attribute 'pack_mode' := '4'}
{attribute 'hide'}
METHOD TcQueryInterface : HRESULT
VAR_INPUT
	iid	: REFERENCE TO IID;
	pipItf	: POINTER TO PVOID;
END_VAR
VAR
	ipSink : ITcIoBACnetServiceResponseSink;
	ipUnknown : ITcUnknown;	
END_VAR
IF GuidsEqual(ADR(iid), ADR(TC_GLOBAL_IID_LIST.IID_ITcIoBACnetServiceResponseSink)) THEN
	ipSink := THIS^; // cast to interface pointer
	pipItf^ := ITCUNKNOWN_TO_PVOID(ipSink);
	TcAddRef();
	TcQueryInterface := S_OK;
ELSIF GuidsEqual(ADR(iid), ADR(TC_GLOBAL_IID_LIST.IID_ITcUnknown)) THEN
	ipUnknown := THIS^; // cast to interface pointer
	pipItf^ := ITCUNKNOWN_TO_PVOID(ipUnknown);
	TcAddRef();
	TcQueryInterface := S_OK;
ELSE
	TcQueryInterface := E_HRESULTAdsErr.NOINTERFACE ; //Call super if this fb extends some other
END_IF
END_METHOD

{attribute 'c++_compatible'}
{attribute 'minimal_input_size' := '4'}
{attribute 'pack_mode' := '4'}
{attribute 'hide'}
METHOD TcRelease : UDINT
END_METHOD

METHOD PRIVATE UpdateTimeStamp : BOOL
VAR_INPUT
END_VAR
IF Valid THEN
	readTsReq(Client := Client, iObject:=iObject, ePropID:=E_BACnetPropIdentifier.PropEventTimeStamps, pData:=ADR(eventTs), nData:=SIZEOF(eventTs));
	readTsReq.Send();
ELSE
	// (BETA) ... Output Error
END_IF
END_METHOD

METHOD GetRequestType : E_BACnetRM_RequestType
VAR_INPUT
END_VAR
GetRequestType := E_BACnetRM_RequestType.eAcknowledge;
END_METHOD

METHOD IsReady : BOOL
VAR_INPUT
END_VAR
IsReady := bReady;
END_METHOD

END_FUNCTION_BLOCK

// POUs/Remote/Requests/[Internal]/FB_BACnetRM_ReqListAdd
{attribute 'c++_compatible'}
{attribute 'enable_dynamic_creation'}
{attribute 'hide'}
FUNCTION_BLOCK FB_BACnetRM_ReqListAdd EXTENDS FB_BACnetRM_ReqBasic
VAR_INPUT
	ePropID : E_BACnetPropIdentifier;
	pData : PVOID;
	nData : UDINT;
END_VAR
VAR 
	req : SendDataRequest;
END_VAR

IF NOT __ISVALIDREF(Client) THEN
	bError:=TRUE;
END_IF

SUPER^();

{attribute 'hide'}
METHOD Send : BOOL
IF Valid THEN
	IF stReq = 0 THEN
		req.service := E_BACnetConfirmedService.SrvAddListElement;
		req.objectIdentifier := iObject.ObjectID;
		req.propertyIdentifier := ePropID;
		req.pData := pData;
		req.nData := nData;
		req.deviceId := Client.ObjectInstance;
		stReq := ADR(req);
	END_IF
	
	Send:=SUPER^.Send();
END_IF
END_METHOD

METHOD PROTECTED ProcessResult : HRESULT
VAR_INPUT
	pResult	: POINTER TO SendDataRequestResult;
END_VAR
bReady:=TRUE;
ProcessResult:=S_OK;
END_METHOD

METHOD GetRequestType : E_BACnetRM_RequestType
VAR_INPUT
END_VAR
GetRequestType := E_BACnetRM_RequestType.eAddListElement;
END_METHOD

METHOD IsReady : BOOL
VAR_INPUT
END_VAR
IsReady := bReady;
END_METHOD

END_FUNCTION_BLOCK

// POUs/Remote/Requests/[Internal]/FB_BACnetRM_ReqListRem
{attribute 'c++_compatible'}
{attribute 'enable_dynamic_creation'}
{attribute 'hide'}
FUNCTION_BLOCK FB_BACnetRM_ReqListRem EXTENDS FB_BACnetRM_ReqBasic
VAR_INPUT
	ePropID : E_BACnetPropIdentifier;
	pData : PVOID;
	nData : UDINT;
END_VAR
VAR 
	req : SendDataRequest;
END_VAR

IF NOT __ISVALIDREF(Client) THEN
	bError:=TRUE;
END_IF

SUPER^();

{attribute 'hide'}
METHOD Send : BOOL
IF Valid THEN
	IF stReq = 0 THEN
		req.service := E_BACnetConfirmedService.SrvRemoveListElement;
		req.objectIdentifier := iObject.ObjectID;
		req.propertyIdentifier := ePropID;
		req.pData := pData;
		req.nData := nData;
		req.deviceId := Client.ObjectInstance;
		stReq := ADR(req);
	END_IF
	
	Send:=SUPER^.Send();
END_IF
END_METHOD

METHOD PROTECTED ProcessResult : HRESULT
VAR_INPUT
	pResult	: POINTER TO SendDataRequestResult;
END_VAR
bReady:=TRUE;
ProcessResult:=S_OK;
END_METHOD

METHOD GetRequestType : E_BACnetRM_RequestType
VAR_INPUT
END_VAR
GetRequestType := E_BACnetRM_RequestType.eRemoveListElement;
END_METHOD

END_FUNCTION_BLOCK

// TEST/TestPackage/Samples/Objects/Local/FB_BACnet_SmplAV01
// [Sample] How to modify Properties (WriteProtect, Disable)?
{attribute 'enable_dynamic_creation'}
FUNCTION_BLOCK FB_BACnet_SmplAV01 EXTENDS FB_BACnet_AV

SUPER^();

METHOD PROTECTED OnObjectStateChanged
SUPER^.OnObjectStateChanged();

CASE (tState) OF
	TCOM_STATE.TCOM_STATE_PREOP:
		// Sample: Disable Properties
		EnableProperty(E_BACnetPropIdentifier.PropUnits, FALSE);
		
		// Sample: WriteProtect Properties
		WriteProtectProperty(E_BACnetPropIdentifier.PropObjectName, TRUE);
		
END_CASE
END_METHOD

END_FUNCTION_BLOCK

// TEST/TestPackage/Samples/Objects/Local/FB_BACnet_SmplBO01
// [Sample] How to implement a process feedback value.
FUNCTION_BLOCK FB_BACnet_SmplBO01 EXTENDS FB_BACnet_BO_IO
VAR_INPUT
	bValFeedback			: BOOL;
END_VAR

SUPER^();

_bFeedbackValue := bValFeedback;

END_FUNCTION_BLOCK

// TEST/TestPackage/Samples/Objects/Remote/FB_BACnetRM_SmplAV01
// [Symple] Sync additional Properties
{attribute 'enable_dynamic_creation'}
FUNCTION_BLOCK FB_BACnetRM_SmplAV01 EXTENDS FB_BACnetRM_AV
VAR_OUTPUT
	eActivePrio		: E_BACnet_Priority;
END_VAR

SUPER^();

METHOD PROTECTED OnObjectStateChanged
SUPER^.OnObjectStateChanged();

// Sync additional properties:
SyncProperty(E_BACnetPropIdentifier.PropCurrentlyActivePriority, SIZEOF(eActivePrio), ADR(eActivePrio), E_BA_SyncModeRM.eRead);
END_METHOD

END_FUNCTION_BLOCK

// TEST/TestPackage/Samples/Project Structure/PRG02/TEMPLATES/Custom/H/HtgCirABC123/FB_BA_HtgCirABC123
FUNCTION_BLOCK FB_BA_HtgCirABC123 EXTENDS FB_BACnet_View
VAR_INPUT CONSTANT
	WthT							: FB_BACnet_AI_IO := (
										iParent 					:= THIS^,
										sObjectName					:= '\/WTHT',
										sDescription				:= '\/Aussentemperatur',
										sDeviceType					:= 'Temperatursensor',
										fResolution					:= 0.003051851,
										eUnit						:= E_BA_Unit.eTemperature_DegreesCelsius);
										
	FlWT							: FB_BACnet_AI_IO := (
										iParent 					:= THIS^,
										sObjectName					:= '\/TVL',
										sDescription				:= '\/Vorlauftemperatur',
										sDeviceType					:= 'Temperatursensor',
										fResolution					:= 0.003051851,
										eUnit						:= E_BA_Unit.eTemperature_DegreesCelsius);
	RtWT							: FB_BACnet_AI_IO := (
										iParent 					:= THIS^,
										sObjectName					:= '\/TRT',
										sDescription				:= '\/Rücklauftemperatur',
										sDeviceType					:= 'Temperatursensor',
										fResolution					:= 0.003051851,
										fScaleOffset				:= 0,
										eUnit						:= E_BA_Unit.eTemperature_DegreesCelsius);
										
	Sched							: FB_BACnet_SchedB := (
										iParent 					:= THIS^,
										sObjectName					:= '\/SCH01',
										sDescription				:= '\/Zeitschaltprogramm',
										aWeek						:= F_BACnet_SchedWeekly3xB(E_BA_Weekday.eMonday, E_BA_Weekday.eFriday, T#0H, FALSE, T#6H, TRUE, T#20H, FALSE));
										
	PID								: FB_BACnet_Loop := (
										iParent 					:= THIS^,
										sObjectName					:= '\/PID01',
										sDescription				:= '\/Vorlauftemperatirregler',
										eAction						:= E_BA_Action.eReverse,
										fProportionalConstant		:= 1,
										fIntegralConstant			:= 180);	
										
	OpM								: FB_Bnet_H_OpM := (
										iParent 					:= THIS^);	
										
	SpG								: FB_Bnet_H_HtgCir_Sp := (
										iParent 					:= THIS^);	
										
	HtgLimit						: FB_Bnet_H_HtgCir_HtgLmt := (
										iParent 					:= THIS^);
										
	Vlv								: FB_Bnet_Vlv_013 := (
										iParent 					:= THIS^);	
										
	Pu								: FB_Bnet_Pu1st := (
										iParent 					:= THIS^);	
END_VAR
VAR // added by the converter: edge detectors and wires of the graphical bodies
    _w1 : ANY;
END_VAR

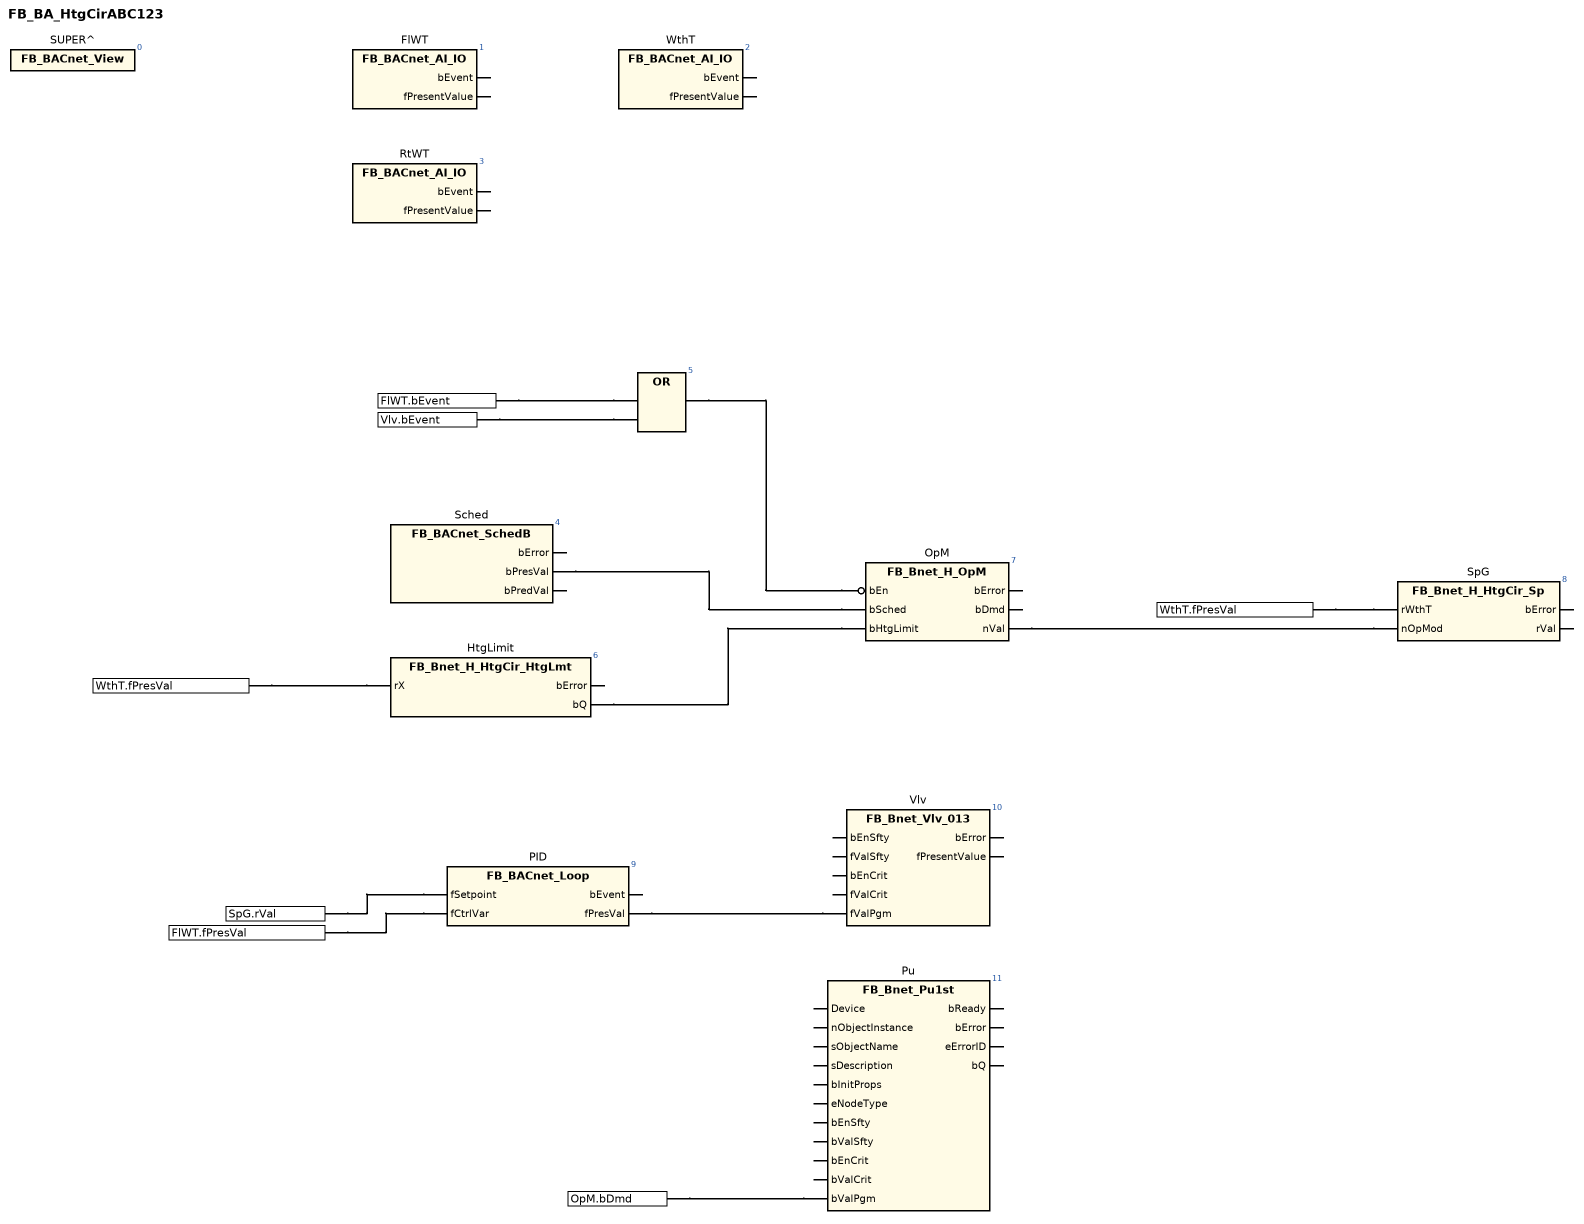
// note: 28 stored wires end on pins the file does not list and are not shown
SUPER^(); // FB_BACnet_View
FlWT(); // FB_BACnet_AI_IO
WthT(); // FB_BACnet_AI_IO
RtWT(); // FB_BACnet_AI_IO
Sched(); // FB_BACnet_SchedB
_w1 := FlWT.bEvent OR Vlv.bEvent;
HtgLimit(rX := WthT.fPresVal); // FB_Bnet_H_HtgCir_HtgLmt
OpM(bEn := NOT _w1, bSched := Sched.bPresVal, bHtgLimit := HtgLimit.bQ); // FB_Bnet_H_OpM
SpG(rWthT := WthT.fPresVal, nOpMod := OpM.nVal); // FB_Bnet_H_HtgCir_Sp
PID(fSetpoint := SpG.rVal, fCtrlVar := FlWT.fPresVal); // FB_BACnet_Loop
Vlv(fValPgm := PID.fPresVal); // FB_Bnet_Vlv_013
Pu(bValPgm := OpM.bDmd); // FB_Bnet_Pu1st

METHOD FB_init : BOOL
VAR_INPUT
	bInitRetains : BOOL; // if TRUE, the retain variables are initialized (warm start / cold start)
	bInCopyCode : BOOL;  // if TRUE, the instance afterwards gets moved into the copy code (online change)
END_VAR
sObjectName		:= '\/HCR01';
sDescription	:= '\/Heizkreis';

Pu.BO.sObjectName := '\/XXXtest';
END_METHOD

END_FUNCTION_BLOCK

// TEST/TestPackage/Templates/HeatSupply/HeatingCircuit/FB_Bnet_H_HtgCir_HtgLmt
FUNCTION_BLOCK FB_Bnet_H_HtgCir_HtgLmt EXTENDS FB_BACnet_View
VAR_INPUT
	rX			: REAL;// Istwert	// Actual value
END_VAR
VAR_OUTPUT
	bQ			: BOOL;// Heizgrenzschalter Schaltbefehl Ein/Aus	// Heating limit switching command on/off
END_VAR
VAR
	Sp								:	FB_BACnet_AV_Setp := (
											iParent 			:= THIS^,
											sObjectName			:= '\/SP01',
											sDescription		:= '\/Sollwert',
											eUnit				:= E_BA_Unit.eTemperature_DegreesCelsius,
											fValue				:= 15.0);
											
	
	Hys				:	FB_Swi2P;//Hysterese Heizgrenze//Hysteresis heating limit
	
	Q								:	FB_BACnet_BV_Disp := (
											iParent 			:= THIS^,
											sObjectName			:= '\/STA01',
											sDescription		:= '\/Status',
											sActiveText			:= 'Ein',
											sInactiveText		:= 'Aus');
END_VAR
VAR // added by the converter: edge detectors and wires of the graphical bodies
    _w1, _w2 : ANY;
END_VAR

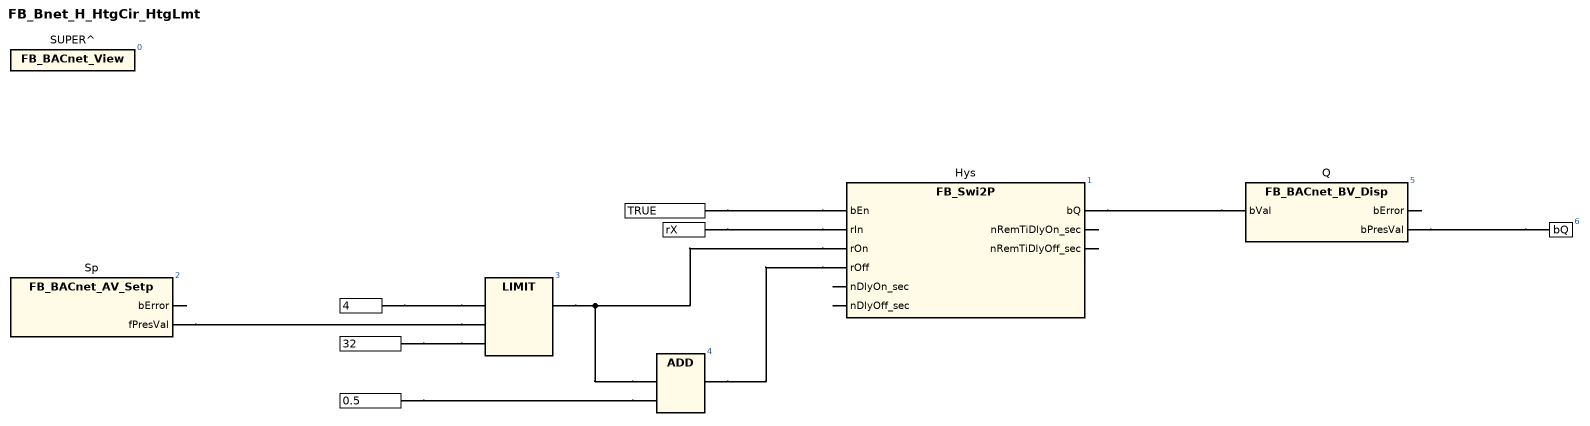
// note: 4 stored wires end on pins the file does not list and are not shown
SUPER^(); // FB_BACnet_View
Hys(bEn := TRUE, rIn := rX, rOn := _w1, rOff := _w2); // FB_Swi2P
Sp(); // FB_BACnet_AV_Setp
_w1 := LIMIT(4, Sp.fPresVal, 32);
_w2 := _w1 + 0.5;
Q(bVal := Hys.bQ); // FB_BACnet_BV_Disp
bQ := Q.bPresVal;

METHOD FB_init : BOOL
VAR_INPUT
	bInitRetains : BOOL; // if TRUE, the retain variables are initialized (warm start / cold start)
	bInCopyCode : BOOL;  // if TRUE, the instance afterwards gets moved into the copy code (online change)
END_VAR
sObjectName		:= '\/GW01';
sDescription	:= '\/Heizgrenzwert';
END_METHOD

END_FUNCTION_BLOCK

// TEST/TestPackage/Templates/HeatSupply/HeatingCircuit/FB_Swi2P
FUNCTION_BLOCK FB_Swi2P
VAR_INPUT
	bEn            : BOOL;// FB-enable
	rIn            : REAL;// input-value
	rOn            : REAL;// Switch-on point
	rOff           : REAL;// Switch-off point
	nDlyOn_sec		: UDINT;// (0..Const.nTiSec) switch-on delay [s]
	nDlyOff_sec		: UDINT;// (0..Const.nTiSec) switch-off delay [s]
END_VAR
VAR_OUTPUT
	bQ                 : BOOL;// control output
	nRemTiDlyOn_sec   : UDINT;// switch-on delay countdown [s]
	nRemTiDlyOff_sec  : UDINT;// switch-off delay countdown [s]
END_VAR
VAR
	tDlyOn				: TIME;
	tDlyOff				: TIME;
	tonDlyOn			: TON;
	tonDlyOff			: TON;
	rtrig				: R_TRIG;
	ftrig				: F_TRIG;
END_VAR

tDlyOn := TO_TIME(1000 * nDlyOn_sec);
tDlyOff := TO_TIME(1000 * nDlyOff_sec);

IF	bEn
THEN
	rtrig(CLK := rOn >= rOff);
	ftrig(CLK := rOn >= rOff);

	IF	rtrig.Q OR
		ftrig.Q
	THEN
		tonDlyOn(IN:= FALSE, PT:= T#0s);
		tonDlyOff(IN:= FALSE, PT:= T#0s);
		bQ := FALSE;
	END_IF

	IF	rOn >= rOff
	THEN
		IF	rOn = rOff
		THEN
			tonDlyOn(IN:= rIn >= rOn, PT:= tDlyOn);

			IF	tonDlyOn.Q
			THEN
				bQ := TRUE;
			END_IF

			tonDlyOff(IN:= bQ AND rIn < rOff, PT:= tDlyOff);

			IF	tonDlyOff.Q
			THEN
				bQ := FALSE;
			END_IF
		ELSE
			tonDlyOn(IN:= rIn >= rOn, PT:= tDlyOn);

			IF	tonDlyOn.Q
			THEN
				bQ := TRUE;
			END_IF

			tonDlyOff(IN:= bQ AND rIn <= rOff, PT:= tDlyOff);

			IF	tonDlyOff.Q
			THEN
				bQ := FALSE;
			END_IF
		END_IF
	ELSE
		tonDlyOn(IN:= rIn <= rOn, PT:= tDlyOn);

		IF	tonDlyOn.Q
		THEN
			bQ := TRUE;
		END_IF

		tonDlyOff(IN:= bQ AND rIn >= rOff, PT:= tDlyOff);

		IF	tonDlyOff.Q
		THEN
			bQ := FALSE;
		END_IF
	END_IF

	nRemTiDlyOn_sec := F_RemSecsTon(tonTimer := tonDlyOn);
	nRemTiDlyOff_sec := F_RemSecsTon(tonTimer := tonDlyOff);
ELSE
	tonDlyOn(IN:= FALSE, PT:= T#0s);
	tonDlyOff(IN:= FALSE, PT:= T#0s);
	nRemTiDlyOn_sec := nRemTiDlyOff_sec := 0;
	bQ := FALSE;
END_IF

END_FUNCTION_BLOCK

// TEST/TestPackage/Templates/Universal/AntiBlocking/F_RemSecsTon
{attribute 'hide'}
FUNCTION F_RemSecsTon : UDINT
VAR_INPUT
	tonTimer			: TON;		// Input of TON-Timer to be evaluated
END_VAR
VAR
	nRemTime_sec		: UDINT;		// remaining time in seconds of TP-Timeer
END_VAR

(*showing remaining Seconds of a timer
with +1-correction and 0, if timer is NOT running*)

nRemTime_sec	:= TO_UDINT((tonTimer.PT-tonTimer.ET)/1000)+1;

IF nRemTime_sec > TO_UDINT((tonTimer.PT)/1000) 		THEN
	nRemTime_sec := TO_UDINT((tonTimer.PT)/1000);
END_IF

IF tonTimer.Q		THEN
	nRemTime_sec := 0;
END_IF

F_RemSecsTon:=nRemTime_sec;

END_FUNCTION

// TEST/TestPackage/Templates/HeatSupply/FB_Bnet_H_OpM
FUNCTION_BLOCK FB_Bnet_H_OpM EXTENDS FB_BACnet_View
VAR_INPUT
	bEn				: BOOL;		//	Freigabe Betrieb							// Release operation
	bSched			: BOOL;		//	Zeitschaltplan Comfort und Economy Betrieb	// Switching schedule Comfort and Economy operation
	bHtgLimit		: BOOL;		// 	Heizgrenzschalter Schaltbefehl Ein/Aus		// Heating limit switching command on/off	
END_VAR
VAR_OUTPUT
	bDmd			: BOOL;		// 	Freigabe Heizkreis/Anforderung Wärmebedarf	// Enable heating circuit/requirement heat demand
	nVal			: UDINT;	// 	Betriebsart Protection,Economy,Comfort 		// Operating mode Protection,Economy,Comfort
END_VAR
VAR
	Man								:	FB_BACnet_MV_Setp := (
											iParent 			:= THIS^,
											sObjectName			:= '\/BAM01',
											sDescription		:= '\/Manuelle Betriebsart',
											sStateText			:= [ 'Auto', 'Schutzbetrieb', 'Economy', 'Comfort' ],
											nValue				:= 1);
											
	OpModPrioSwi				: FB_PrioSwi_UDI08;	//	Priorisierung Betriebsart	//	Prioritization operating mode

	PrOp							:	FB_BACnet_MV_Disp := (
											iParent 			:= THIS^,
											sObjectName			:= '\/BAS01',
											sDescription		:= '\/Aktuelle Betriebsart',
											sStateText			:= [ 'Schutzbetrieb', 'Economy', 'Comfort' ]);
											

	DmdPrioSwi					: FB_PrioSwi_B04;//Priorisierung Anforderung Wärmebedarf//Prioritization requirement heat demand

	Dmd								:	FB_BACnet_BV_Disp := (
											iParent 			:= THIS^,
											sObjectName			:= '\/AF01',
											sDescription		:= '\/Anforderung Heizen',
											sActiveText			:= 'Aktiv',
											sInactiveText		:= 'Inaktiv');
END_VAR
VAR // added by the converter: edge detectors and wires of the graphical bodies
    _w1, _w2, _w3, _w4, _w5, _w6 : ANY;
END_VAR

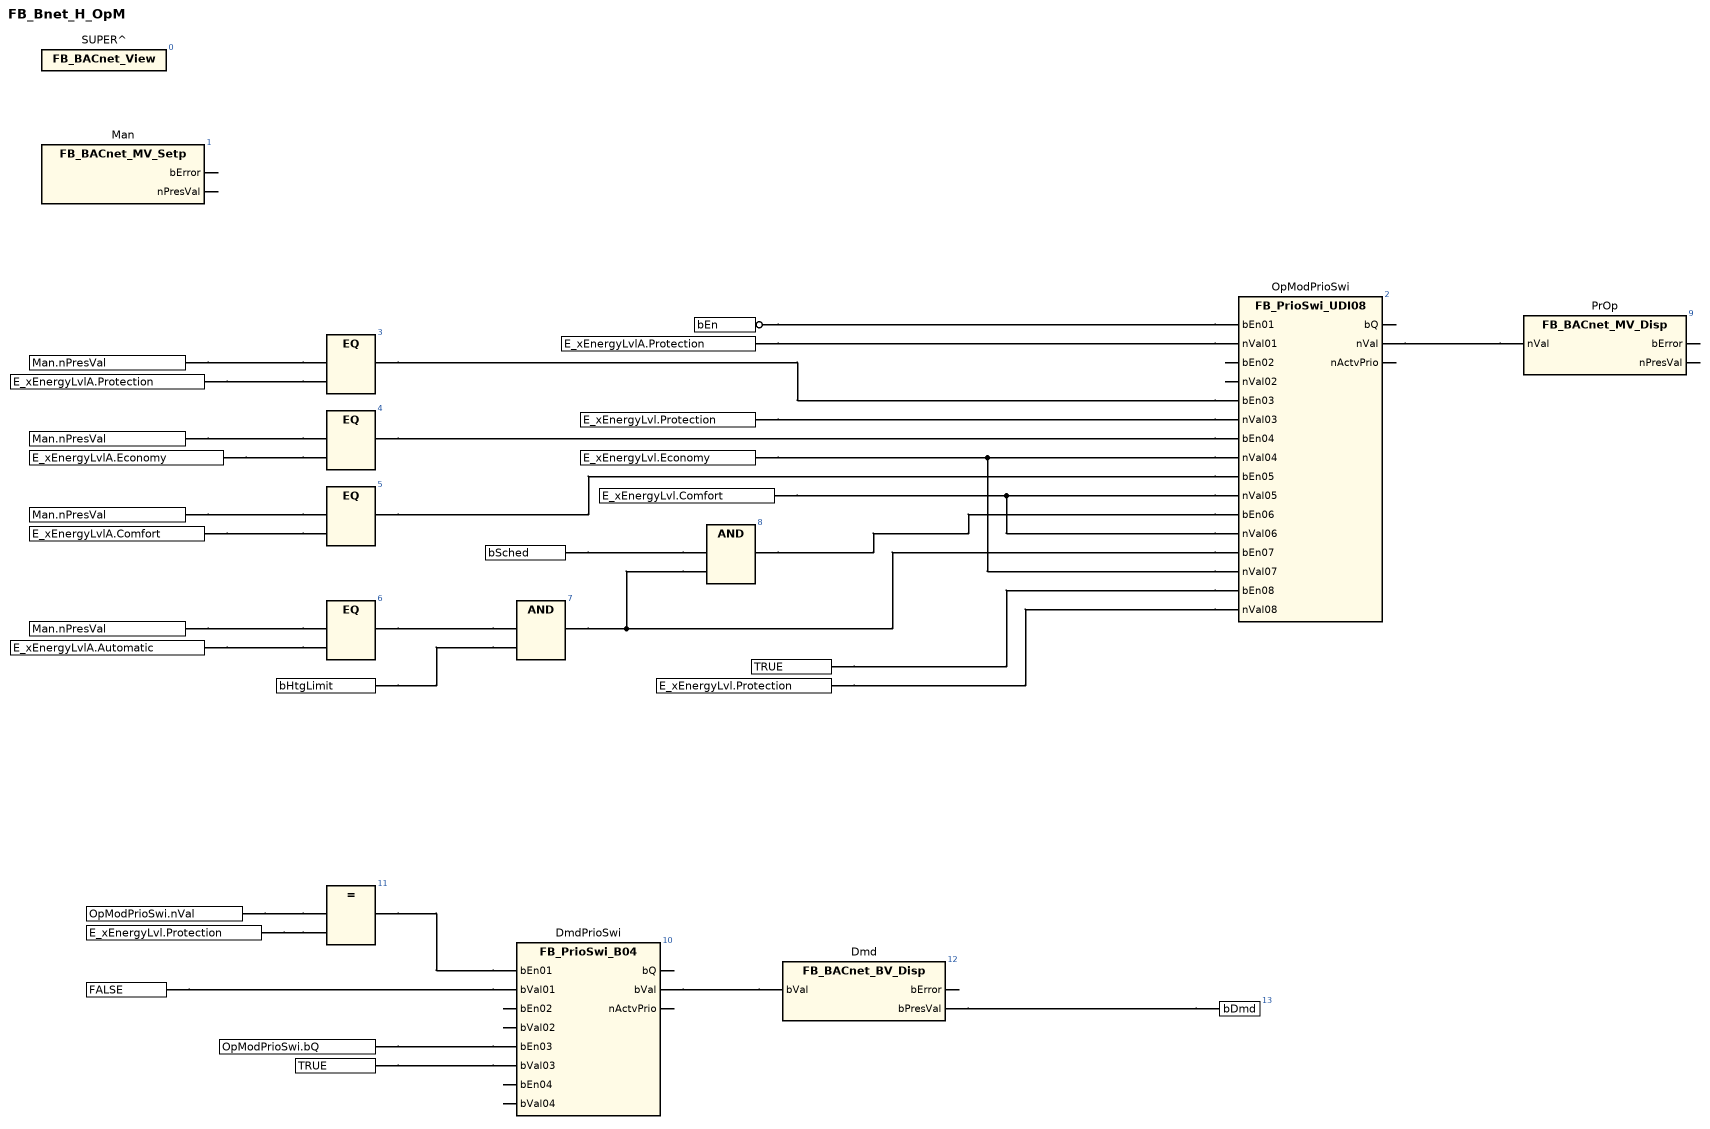
// note: 18 stored wires end on pins the file does not list and are not shown
SUPER^(); // FB_BACnet_View
Man(); // FB_BACnet_MV_Setp
OpModPrioSwi(
    bEn01 := NOT bEn,
    nVal01 := E_xEnergyLvlA.Protection,
    bEn03 := _w1,
    nVal03 := E_xEnergyLvl.Protection,
    bEn04 := _w2,
    nVal04 := E_xEnergyLvl.Economy,
    bEn05 := _w3,
    nVal05 := E_xEnergyLvl.Comfort,
    bEn06 := _w4,
    nVal06 := E_xEnergyLvl.Comfort,
    bEn07 := _w5,
    nVal07 := E_xEnergyLvl.Economy,
    bEn08 := TRUE,
    nVal08 := E_xEnergyLvl.Protection); // FB_PrioSwi_UDI08
_w1 := Man.nPresVal = E_xEnergyLvlA.Protection;
_w2 := Man.nPresVal = E_xEnergyLvlA.Economy;
_w3 := Man.nPresVal = E_xEnergyLvlA.Comfort;
_w5 := Man.nPresVal = E_xEnergyLvlA.Automatic AND bHtgLimit;
_w4 := bSched AND _w5;
PrOp(nVal := OpModPrioSwi.nVal); // FB_BACnet_MV_Disp
DmdPrioSwi(bEn01 := _w6, bVal01 := FALSE, bEn03 := OpModPrioSwi.bQ, bVal03 := TRUE); // FB_PrioSwi_B04
_w6 := OpModPrioSwi.nVal = E_xEnergyLvl.Protection;
Dmd(bVal := DmdPrioSwi.bVal); // FB_BACnet_BV_Disp
bDmd := Dmd.bPresVal;

METHOD FB_init : BOOL
VAR_INPUT
	bInitRetains : BOOL; // if TRUE, the retain variables are initialized (warm start / cold start)
	bInCopyCode : BOOL;  // if TRUE, the instance afterwards gets moved into the copy code (online change)
END_VAR
sObjectName		:= '\/OPM01';
sDescription	:= '\/Betriebsart';
END_METHOD

END_FUNCTION_BLOCK

// TEST/TestPackage/Templates/HeatSupply/FB_PrioSwi_UDI08
FUNCTION_BLOCK FB_PrioSwi_UDI08
VAR_INPUT
	bEn01		: BOOL;		// Enabling the priority value
	nVal01		: UDINT;	// Priority value
	bEn02		: BOOL;		// Enabling the priority value
	nVal02		: UDINT;	// Priority value
	bEn03		: BOOL;		// Enabling the priority value
	nVal03		: UDINT;	// Priority value
	bEn04		: BOOL;		// Enabling the priority value
	nVal04		: UDINT;	// Priority value
	bEn05		: BOOL;		// Enabling the priority value
	nVal05		: UDINT;	// Priority value
	bEn06		: BOOL;		// Enabling the priority value
	nVal06		: UDINT;	// Priority value
	bEn07		: BOOL;		// Enabling the priority value
	nVal07		: UDINT;	// Priority value
	bEn08		: BOOL;		// Enabling the priority value
	nVal08		: UDINT;	// Priority value
END_VAR
VAR_OUTPUT
	bQ			: BOOL;		// Output to indicate whether a priority is enabled
	nVal		: UDINT;	// Output of the value of the current (highest) priority that is enabled
	nActvPrio	: UDINT;		// Current (highest) priority that is enabled
END_VAR
VAR
	aEn			: ARRAY [1..cBA_PrioSwiUDI08] OF BOOL;
	aVal		: ARRAY [1..cBA_PrioSwiUDI08] OF UDINT;
	i			: UDINT;
END_VAR
VAR CONSTANT
	cBA_PrioSwiUDI08    : UDINT := 8;
END_VAR

aEn[1] := bEn01;
aEn[2] := bEn02;
aEn[3] := bEn03;
aEn[4] := bEn04;
aEn[5] := bEn05;
aEn[6] := bEn06;
aEn[7] := bEn07;
aEn[8] := bEn08;

aVal[1] := nVal01;
aVal[2] := nVal02;
aVal[3] := nVal03;
aVal[4] := nVal04;
aVal[5] := nVal05;
aVal[6] := nVal06;
aVal[7] := nVal07;
aVal[8] := nVal08;

bQ := FALSE;
nVal := 0;
nActvPrio := Const.nNoActvPrio;

FOR i := 1 TO cBA_PrioSwiUDI08 BY 1 DO
	IF	aEn[i] = TRUE
	THEN
		bQ := TRUE;
		nVal := aVal[i];
		nActvPrio := i;
		EXIT;
	END_IF
END_FOR

END_FUNCTION_BLOCK

// TEST/TestPackage/Templates/HeatSupply/FB_PrioSwi_B04
FUNCTION_BLOCK FB_PrioSwi_B04
VAR_INPUT
	bEn01		: BOOL;	// Enabling the priority value
	bVal01		: BOOL;	// Priority value
	bEn02		: BOOL;	// Enabling the priority value
	bVal02		: BOOL;	// Priority value
	bEn03		: BOOL;	// Enabling the priority value
	bVal03		: BOOL;	// Priority value
	bEn04		: BOOL;	// Enabling the priority value
	bVal04		: BOOL;	// Priority value
END_VAR
VAR_OUTPUT
	bQ			: BOOL;	// Output to indicate whether a priority is enabled
	bVal		: BOOL;	// Output of the value of the current (highest) priority that is enabled
	nActvPrio	: UDINT;	// Current (highest) priority that is enabled
END_VAR
VAR
	aEn			: ARRAY [1..cBA_PrioSwiB04] OF BOOL;
	aVal		: ARRAY [1..cBA_PrioSwiB04] OF BOOL;
	i			: UDINT;
END_VAR
VAR CONSTANT
	cBA_PrioSwiB04    : UDINT := 4;
END_VAR

aEn[1] := bEn01;
aEn[2] := bEn02;
aEn[3] := bEn03;
aEn[4] := bEn04;

aVal[1] := bVal01;
aVal[2] := bVal02;
aVal[3] := bVal03;
aVal[4] := bVal04;

bQ := FALSE;
bVal := FALSE;
nActvPrio := Const.nNoActvPrio;

FOR i := 1 TO cBA_PrioSwiB04 BY 1 DO
	IF	aEn[i] = TRUE
	THEN
		bQ := TRUE;
		bVal := aVal[i];
		nActvPrio := i;
		EXIT;
	END_IF
END_FOR

END_FUNCTION_BLOCK

// TEST/TestPackage/Templates/HeatSupply/HeatingCircuit/FB_Bnet_H_HtgCir_Sp
FUNCTION_BLOCK FB_Bnet_H_HtgCir_Sp EXTENDS FB_BACnet_View
VAR_INPUT
	rWthT			: REAL;
	nOpMod		: UDINT;	// Betriebsart	// Operating mode 
END_VAR
VAR_INPUT CONSTANT PERSISTENT
	HeatingSetpointProtection : REAL := 5;
END_VAR
VAR_OUTPUT
	rVal			: REAL;	//Sollwert Heizkreis//Setpoint heating circuit	
END_VAR
VAR_INPUT CONSTANT
	Curve							:	FB_Bnet_Scale_04 := (
											iParent			:= THIS^);
										
	NightOffs						:	FB_BACnet_AV_Setp := (
											iParent 			:= THIS^,
											sObjectName			:= '\/SP01',
											sDescription		:= '\/Sollwert Nachtabsenkung',
											eUnit				:= E_BA_Unit.eTemperature_DegreesCelsius,
											fValue				:= 8.0);

	SpFlWT							:	FB_BACnet_AV_Disp := (
											iParent 			:= THIS^,
											sObjectName			:= '\/SWC01',
											sDescription		:= '\/Errechnete Vorlauftemperatur',
											eUnit				:= E_BA_Unit.eTemperature_DegreesCelsius);
END_VAR
VAR
	PrioSwi			:	FB_MMUX_R04;//Priorisierung des Sollwertes//Prioritization of the setpoint
END_VAR
VAR // added by the converter: edge detectors and wires of the graphical bodies
    _w1 : ANY;
END_VAR

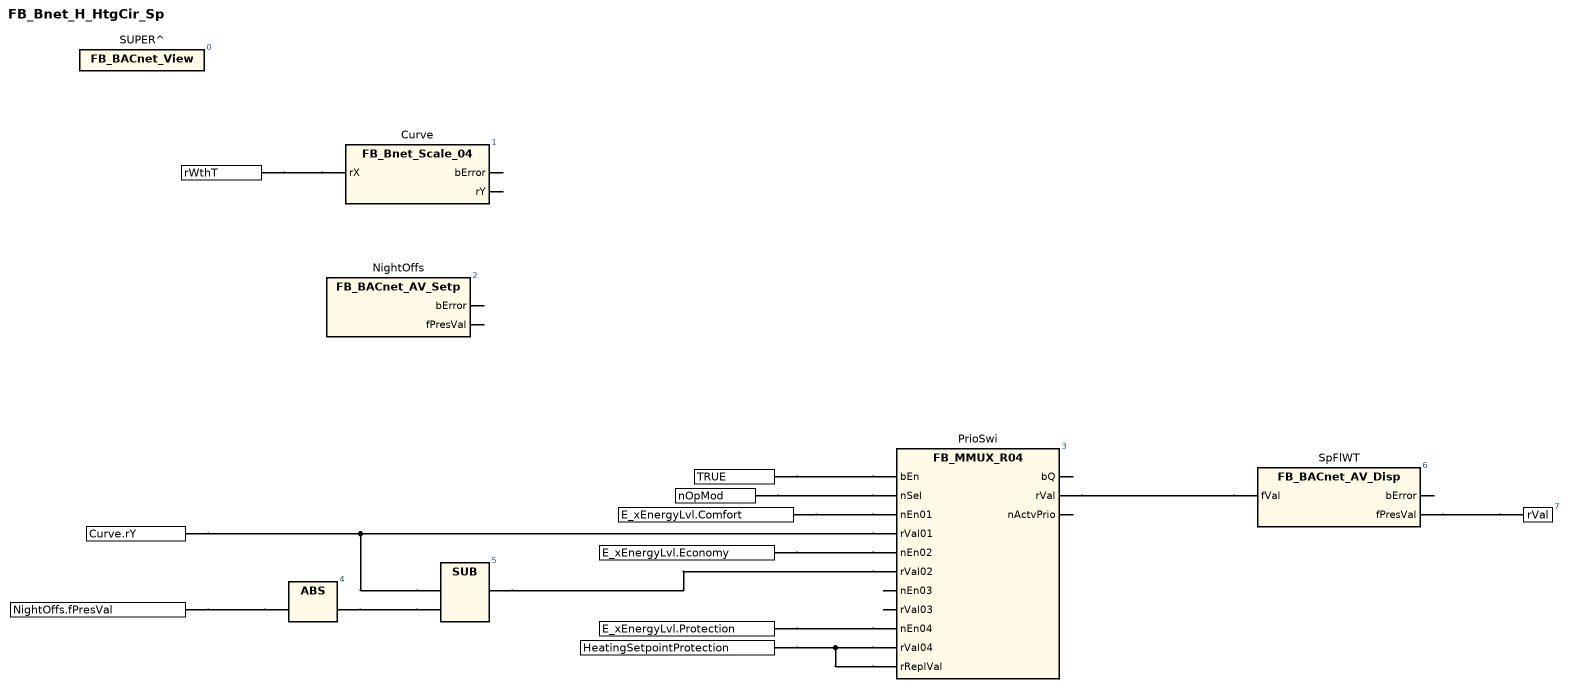
// note: 10 stored wires end on pins the file does not list and are not shown
SUPER^(); // FB_BACnet_View
Curve(rX := rWthT); // FB_Bnet_Scale_04
NightOffs(); // FB_BACnet_AV_Setp
PrioSwi(
    bEn := TRUE,
    nSel := nOpMod,
    nEn01 := E_xEnergyLvl.Comfort,
    rVal01 := Curve.rY,
    nEn02 := E_xEnergyLvl.Economy,
    rVal02 := _w1,
    nEn04 := E_xEnergyLvl.Protection,
    rVal04 := HeatingSetpointProtection,
    rReplVal := HeatingSetpointProtection); // FB_MMUX_R04
_w1 := Curve.rY - ABS(NightOffs.fPresVal);
SpFlWT(fVal := PrioSwi.rVal); // FB_BACnet_AV_Disp
rVal := SpFlWT.fPresVal;

METHOD FB_init : BOOL
VAR_INPUT
	bInitRetains : BOOL; // if TRUE, the retain variables are initialized (warm start / cold start)
	bInCopyCode : BOOL;  // if TRUE, the instance afterwards gets moved into the copy code (online change)
END_VAR
sObjectName		:= '\/SP01';
sDescription	:= '\/Sollwerte';
END_METHOD

END_FUNCTION_BLOCK

// TEST/TestPackage/Templates/Universal/Control/Scale/FB_Bnet_Scale_04
FUNCTION_BLOCK FB_Bnet_Scale_04 EXTENDS FB_BACnet_View
VAR_INPUT
	rX			:	REAL;	//	Istwert	//	Actual value
END_VAR
VAR_OUTPUT
	rY			:	REAL;	//	Skalierter Wert	//	scaled value
END_VAR
VAR
//Skalierung mit 4 Stützpunkten//Scaling with 4 interpolation points

	X1								:	FB_BACnet_AV_Setp := (
											iParent 			:= THIS^,
											sObjectName			:= '\/STX01',
											sDescription		:= '\/Stützpunkt X1',
											eUnit				:= E_BA_Unit.eTemperature_DegreesCelsius,
											fValue				:= 15);
	X2								:	FB_BACnet_AV_Setp := (
											iParent 			:= THIS^,
											sObjectName			:= '\/STX02',
											sDescription		:= '\/Stützpunkt X2',
											eUnit				:= E_BA_Unit.eTemperature_DegreesCelsius,
											fValue				:= 5);
	X3								:	FB_BACnet_AV_Setp := (
											iParent 			:= THIS^,
											sObjectName			:= '\/STX03',
											sDescription		:= '\/Stützpunkt X3',
											eUnit				:= E_BA_Unit.eTemperature_DegreesCelsius,
											fValue				:= 0);
	X4								:	FB_BACnet_AV_Setp := (
											iParent 			:= THIS^,
											sObjectName			:= '\/STX04',
											sDescription		:= '\/Stützpunkt X4',
											eUnit				:= E_BA_Unit.eTemperature_DegreesCelsius,
											fValue				:= -15);
											
	Y1								:	FB_BACnet_AV_Setp := (
											iParent 			:= THIS^,
											sObjectName			:= '\/STY01',
											sDescription		:= '\/Stützpunkt Y1',
											eUnit				:= E_BA_Unit.eTemperature_DegreesCelsius,
											fValue				:= 21);
	Y2								:	FB_BACnet_AV_Setp := (
											iParent 			:= THIS^,
											sObjectName			:= '\/STY02',
											sDescription		:= '\/Stützpunkt Y2',
											eUnit				:= E_BA_Unit.eTemperature_DegreesCelsius,
											fValue				:= 35);
	Y3								:	FB_BACnet_AV_Setp := (
											iParent 			:= THIS^,
											sObjectName			:= '\/STY03',
											sDescription		:= '\/Stützpunkt Y3',
											eUnit				:= E_BA_Unit.eTemperature_DegreesCelsius,
											fValue				:= 45);
	Y4								:	FB_BACnet_AV_Setp := (
											iParent 			:= THIS^,
											sObjectName			:= '\/STY04',
											sDescription		:= '\/Stützpunkt Y4',
											eUnit				:= E_BA_Unit.eTemperature_DegreesCelsius,
											fValue				:= 65);


	Scale			: FB_Chrct04;//Skalierungsfunktion//scaling function
	
	CalcSp							:	FB_BACnet_AV_Disp := (
											iParent 			:= THIS^,
											sObjectName			:= '\/CSP01',
											sDescription		:= '\/Errechneter Sollwert',
											eUnit				:= E_BA_Unit.eTemperature_DegreesCelsius);
END_VAR

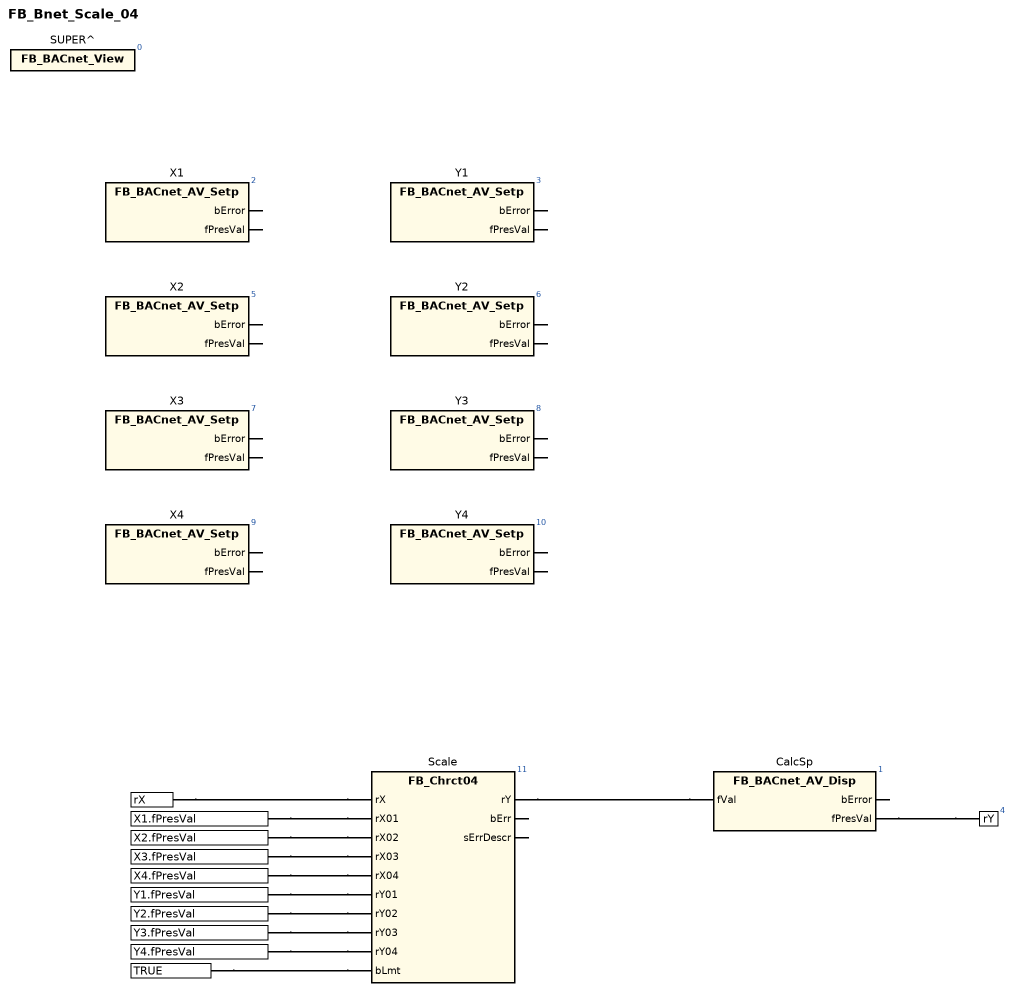
SUPER^(); // FB_BACnet_View
CalcSp(fVal := Scale.rY); // FB_BACnet_AV_Disp
X1(); // FB_BACnet_AV_Setp
Y1(); // FB_BACnet_AV_Setp
rY := CalcSp.fPresVal;
X2(); // FB_BACnet_AV_Setp
Y2(); // FB_BACnet_AV_Setp
X3(); // FB_BACnet_AV_Setp
Y3(); // FB_BACnet_AV_Setp
X4(); // FB_BACnet_AV_Setp
Y4(); // FB_BACnet_AV_Setp
Scale(
    rX := rX,
    rX01 := X1.fPresVal,
    rX02 := X2.fPresVal,
    rX03 := X3.fPresVal,
    rX04 := X4.fPresVal,
    rY01 := Y1.fPresVal,
    rY02 := Y2.fPresVal,
    rY03 := Y3.fPresVal,
    rY04 := Y4.fPresVal,
    bLmt := TRUE); // FB_Chrct04

METHOD FB_init : BOOL
VAR_INPUT
	bInitRetains : BOOL; // if TRUE, the retain variables are initialized (warm start / cold start)
	bInCopyCode : BOOL;  // if TRUE, the instance afterwards gets moved into the copy code (online change)
END_VAR
sObjectName		:= '\/SCL01';
sDescription	:= '\/Kurve';
END_METHOD

END_FUNCTION_BLOCK

// TEST/TestPackage/Templates/Universal/Control/Scale/FB_Chrct04
FUNCTION_BLOCK FB_Chrct04
VAR_INPUT
	rX			: REAL;	// Input value of the characteristic curve
	rX01		: REAL;	// X-value for interpolation point P1
	rX02		: REAL;	// X-value for interpolation point P2
	rX03		: REAL;	// X-value for interpolation point P3
	rX04		: REAL;	// X-value for interpolation point P4
	rY01		: REAL;	// Y-value for interpolation point P1
	rY02		: REAL;	// Y-value for interpolation point P2
	rY03		: REAL;	// Y-value for interpolation point P3
	rY04		: REAL;	// Y-value for interpolation point P4	
	bLmt		: BOOL;		// True = Limitation lrY in range between Y1 and Y4
END_VAR
VAR_OUTPUT
	rY			: REAL;		// Calculated output value of the characteristic curve
	bErr		: BOOL;			// error
	sErrDescr	: T_MaxString;	// error description
END_VAR
VAR
	aX				: ARRAY [1..cBA_NumOfElem] OF REAL;
	aY				: ARRAY [1..cBA_NumOfElem] OF REAL;
	i				: UDINT;
	rM				: REAL;
	rBuffer1		: REAL;
	rBuffer2		: REAL;
END_VAR

VAR CONSTANT
	cBA_NumOfElem	: UDINT := 4;
END_VAR

	bErr     	:= FALSE;
	sErrDescr	:= '';

	aX[1] := rX01;
	aX[2] := rX02;
	aX[3] := rX03;
	aX[4] := rX04;
	
	aY[1] := rY01;
	aY[2] := rY02;
	aY[3] := rY03;
	aY[4] := rY04;

	FOR i := 1 TO (cBA_NumOfElem - 1) BY 1 DO
		rBuffer1 := aX[i] - aX[i + 1];
		rBuffer2 := 0;
		IF	MEMCMP(pBuf1 := ADR(rBuffer1), pBuf2 := ADR(rBuffer2), n := SIZEOF(rBuffer2)) = 0	THEN
			bErr		:= TRUE;
			sErrDescr	:= '01: Error at entered element no.';
			sErrDescr	:= CONCAT(sErrDescr, TO_STRING(i));
			sErrDescr	:= CONCAT(sErrDescr, '. The following sequence must be adhered to: lrX01 > lrX02 > lrXn OR lrX01 < lrX02 < lrXn');
			rY := 0;
			RETURN;
		END_IF
	END_FOR

(*Berechnung*)
(*X = (Y - Y1) / m + X1*)
	FOR i := 1 TO (cBA_NumOfElem - 1) BY 1 DO
		IF	rX >= aX[i] AND rX <= aX[i + 1] OR rX >= aX[i + 1] AND rX <= aX[i]	THEN
			(*lrM = Steigung*)
			(*m = (Y2 - Y1) / (X2 - X1*)
			rM := (aY[i + 1] - aY[i]) / (aX[i + 1] - aX[i]);
			(*Y = Y1 + m * (X - X1)*)
			rY := aY[i] + rM * (rX - aX[i]);
			RETURN;
		END_IF
	END_FOR

(*Berechnung wenn lrX ausserhalb von aX[1] oder aX[cNumOfEntries] liegt*)
	IF	aX[1] > aX[2] AND aX[1] < rX OR aX[1] < aX[2] AND aX[1] > rX	THEN
		(*lrM = Steigung*)
		(*m = (Y2 - Y1) / (X2 - X1*)
		rM := (rY02 - rY01) / (rX02 - rX01);
		(*Y = Y1 + m * (X - X1)*)
		rY := rY01 + rM * (rX - rX01);
	ELSIF	aX[3] > aX[cBA_NumOfElem] AND aX[cBA_NumOfElem] > rX OR aX[3] < aX[cBA_NumOfElem] AND aX[cBA_NumOfElem] < rX	THEN
		(*lrM = Steigung*)
		(*m = (Y4 - Y3) / (X4 - X3*)
		rM := (rY04 - rY03) / (rX04 - rX03);
		(*Y = Y3 + m * (X - X3)*)
		rY := rY03 + rM * (rX - rX03);
	END_IF

(*Limitierung der Bereichsgrenzen*)
	IF	bLmt	THEN
		IF	aX[1] > aX[2] AND aX[1] < rX OR aX[1] < aX[2] AND aX[1] > rX	THEN
			rY := rY01;
		END_IF
	
		IF	aX[3] > aX[cBA_NumOfElem] AND aX[cBA_NumOfElem] > rX OR aX[3] < aX[cBA_NumOfElem] AND aX[cBA_NumOfElem] < rX	THEN
			rY := rY04;
		END_IF
	END_IF

END_FUNCTION_BLOCK

// TEST/TestPackage/Templates/HeatSupply/HeatingCircuit/FB_MMUX_R04
FUNCTION_BLOCK FB_MMUX_R04
VAR_INPUT
	bEn			: BOOL;	// Activation of the block function
	nSel		: UDINT;// Selector
	nEn01		: UDINT := Const.nNoActvPrio;	// Input selector condition
	rVal01		: REAL;	// Input Value to chose from
	nEn02		: UDINT := Const.nNoActvPrio;	// Input selector condition
	rVal02		: REAL;	// Input Value to chose from
	nEn03		: UDINT := Const.nNoActvPrio;	// Input selector condition
	rVal03		: REAL;	// Input Value to chose from
	nEn04		: UDINT := Const.nNoActvPrio;	// Input selector condition
	rVal04		: REAL;	// Input Value to chose from
	rReplVal	: REAL;	// Substitute value, if no input selector condition is active
END_VAR
VAR_OUTPUT
	bQ			: BOOL;	// TRUE, if the selector nSel matches an input selector condition diNoActvPrio
	rVal		: REAL;	// Value of the selected input selector condition
	nActvPrio  : UDINT;	// Indicates which input selector condition is active
END_VAR

nSel := LIMIT(0,nSel,4294967294);

nActvPrio := Const.nNoActvPrio;
rVal := 0;
bQ := FALSE;

IF	bEn
THEN
	IF	nSel = nEn01
	THEN
		bQ := TRUE;
		rVal := rVal01;
		nActvPrio := 1;
		RETURN;
	END_IF
	
	IF	nSel = nEn02
	THEN
		bQ := TRUE;
		rVal := rVal02;
		nActvPrio := 2;
		RETURN;
	END_IF
	
	IF	nSel = nEn03
	THEN
		bQ := TRUE;
		rVal := rVal03;
		nActvPrio := 3;
		RETURN;
	END_IF
	
	IF	nSel = nEn04
	THEN
		bQ := TRUE;
		rVal := rVal04;
		nActvPrio := 4;
		RETURN;
	END_IF

	rVal := rReplVal;
END_IF

END_FUNCTION_BLOCK

// TEST/TestPackage/Templates/Universal/Valve/FB_Bnet_Vlv_013
FUNCTION_BLOCK FB_Bnet_Vlv_013 EXTENDS FB_BACnet_View
VAR_INPUT
	bEnSfty			: BOOL;
	fValSfty		: REAL;
	bEnCrit			: BOOL;
	fValCrit		: REAL;
	fValPgm			: REAL;
END_VAR
VAR_OUTPUT
	fPresentValue	: REAL;
	bEvent			: BOOL;
END_VAR
VAR
	AO								: FB_BACnet_AO_IO5P := (
										iParent 				:= THIS^,
										sObjectName				:= '\/CMD01',
										sDescription			:= '\/Schaltbefehl',
										sDeviceType				:= 'Ventil',
										fResolution				:= 0.003051851,
										fScaleOffset			:= 0,
										eUnit					:= E_BA_Unit.eOther_Percent);
END_VAR

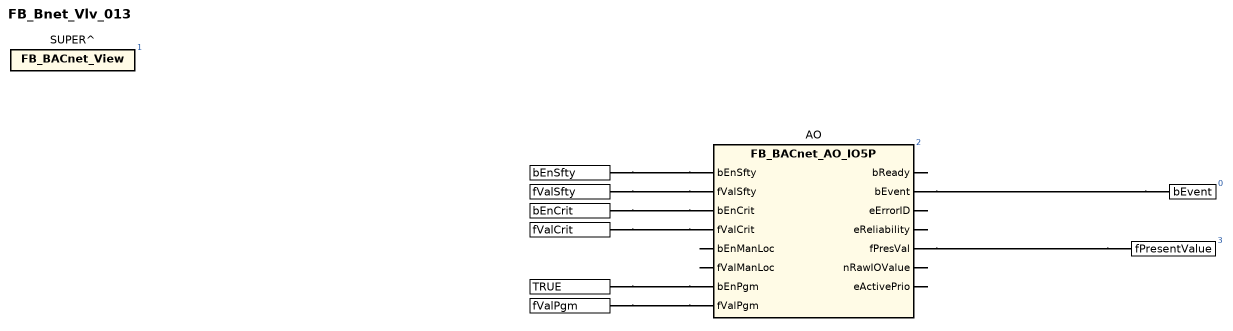
bEvent := AO.bEvent;
SUPER^(); // FB_BACnet_View
AO(
    bEnSfty := bEnSfty,
    fValSfty := fValSfty,
    bEnCrit := bEnCrit,
    fValCrit := fValCrit,
    bEnPgm := TRUE,
    fValPgm := fValPgm); // FB_BACnet_AO_IO5P
fPresentValue := AO.fPresVal;

METHOD FB_init : BOOL
VAR_INPUT
	bInitRetains : BOOL; // if TRUE, the retain variables are initialized (warm start / cold start)
	bInCopyCode : BOOL;  // if TRUE, the instance afterwards gets moved into the copy code (online change)
END_VAR
sObjectName		:= '\/VLV01';
sDescription	:= '\/Ventil';
END_METHOD

END_FUNCTION_BLOCK

// TEST/TestPackage/Templates/Universal/Pump/1st/FB_Bnet_Pu1st
FUNCTION_BLOCK FB_Bnet_Pu1st EXTENDS FB_BACnet_View
VAR_INPUT
	bEnSfty		: BOOL;
	bValSfty	: BOOL;
	bEnCrit		: BOOL;
	bValCrit	: BOOL;
	bValPgm		: BOOL;
END_VAR
VAR_OUTPUT
	bQ			: BOOL;
END_VAR
VAR_INPUT CONSTANT
	Dst								: FB_BACnet_BI_IO := (
										iParent 				:= THIS^,
										sObjectName				:= '\/SM01',
										sDescription			:= '\/Störung',
										sDeviceType				:= 'Sicherung',
										sActiveText				:= 'Ausgelöst',
										sInactiveText			:= 'Normal',
										ePolarity				:= E_BA_Polarity.eReverse,
										nNotificationClass	:= 40,
										aEventEnable			:= [TRUE, TRUE, FALSE]);	
					
	BO								: FB_BACnet_BO_IO5P := (
										iParent 				:= THIS^,
										sObjectName				:= '\/CMD01',
										sDescription			:= '\/Schaltbefehl',
										sDeviceType				:= 'Ausgang',
										sActiveText				:= 'Ein',
										sInactiveText			:= 'Aus');

	DlyOff							: FB_Bnet_DlyOff := (
										iParent 				:= THIS^);

	Ablk							: FB_Bnet_AntiBlocking := (
										iParent 				:= THIS^);
END_VAR
VAR // added by the converter: edge detectors and wires of the graphical bodies
    _w1 : BOOL;
END_VAR

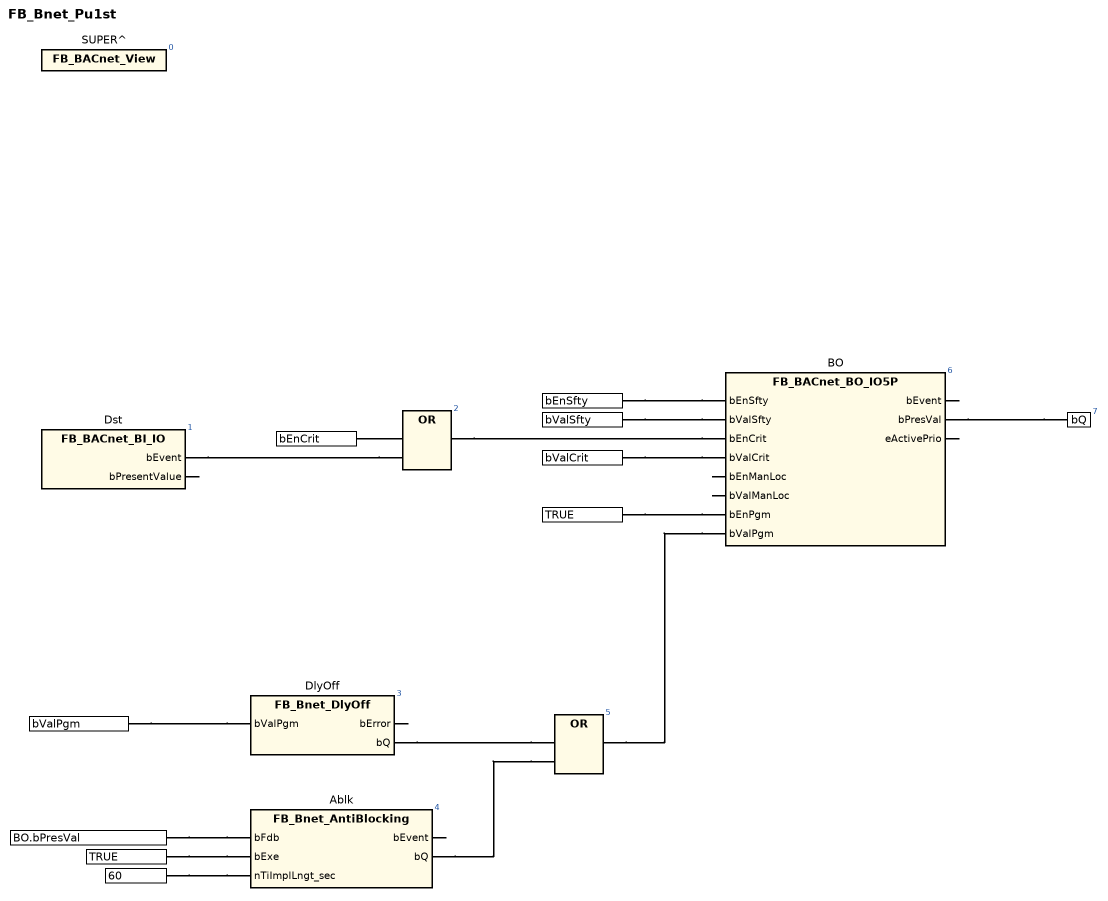
SUPER^(); // FB_BACnet_View
Dst(); // FB_BACnet_BI_IO
_w1 := bEnCrit OR Dst.bEvent;
DlyOff(bValPgm := bValPgm); // FB_Bnet_DlyOff
Ablk(bFdb := BO.bPresVal, bExe := TRUE, nTiImplLngt_sec := 60); // FB_Bnet_AntiBlocking
BO(
    bEnSfty := bEnSfty,
    bValSfty := bValSfty,
    bEnCrit := _w1,
    bValCrit := bValCrit,
    bEnPgm := TRUE,
    bValPgm := DlyOff.bQ OR Ablk.bQ); // FB_BACnet_BO_IO5P
bQ := BO.bPresVal;

METHOD FB_init : BOOL
VAR_INPUT
	bInitRetains : BOOL; // if TRUE, the retain variables are initialized (warm start / cold start)
	bInCopyCode : BOOL;  // if TRUE, the instance afterwards gets moved into the copy code (online change)
END_VAR
sObjectName		:= '\/PU01';
sDescription	:= '\/Pumpe';
END_METHOD

END_FUNCTION_BLOCK

// TEST/TestPackage/Templates/Universal/Control/DelayOff/FB_Bnet_DlyOff
FUNCTION_BLOCK FB_Bnet_DlyOff EXTENDS FB_BACnet_View
VAR_INPUT
	bValPgm		:	BOOL;	//	Wert Programmpriorität		//	Value program priority
END_VAR
VAR_OUTPUT
	bQ			:	BOOL;	//	aktiv	//	active
END_VAR
VAR
	TiVal							:	FB_BACnet_AV_Setp := (
											iParent 			:= THIS^,
											sObjectName			:= '\/SP01',
											sDescription		:= '\/Sollwert',
											eUnit				:= E_BA_Unit.eTime_Seconds,
											fValue				:= 0);
											
	tofDlyOff	: TOF; // Zeitglied Aktor verzögert aus	// Timer actuator delay off
END_VAR

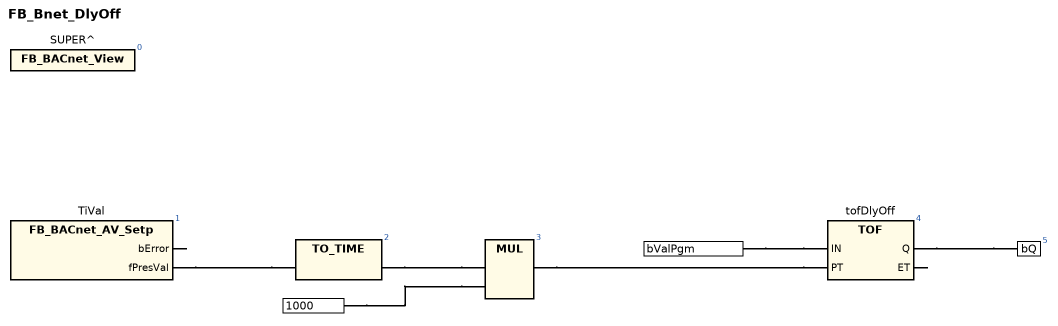
SUPER^(); // FB_BACnet_View
TiVal(); // FB_BACnet_AV_Setp
tofDlyOff(IN := bValPgm, PT := TO_TIME(TiVal.fPresVal) * 1000); // TOF
bQ := tofDlyOff.Q;

METHOD FB_init : BOOL
VAR_INPUT
	bInitRetains : BOOL; // if TRUE, the retain variables are initialized (warm start / cold start)
	bInCopyCode : BOOL;  // if TRUE, the instance afterwards gets moved into the copy code (online change)
END_VAR
sObjectName		:= '\/DLY01';
sDescription	:= '\/Ausschaltverzögerung';
END_METHOD

END_FUNCTION_BLOCK

// TEST/TestPackage/Templates/Universal/AntiBlocking/FB_Bnet_AntiBlocking
FUNCTION_BLOCK FB_Bnet_AntiBlocking EXTENDS FB_BACnet_View
VAR_INPUT CONSTANT PERSISTENT
	bEn				:	BOOL := TRUE;
END_VAR
VAR_INPUT
	bFdb					:	BOOL;	
	bExe					:	BOOL;
	nTiImplLngt_sec			:	UDINT;
END_VAR
VAR_OUTPUT
	bQ			:	BOOL;	//	aktiv	//	active
END_VAR
VAR
	IdlePrd							:	FB_BACnet_AV_Setp := (
											iParent 			:= THIS^,
											sObjectName			:= '\/SP01',
											sDescription		:= '\/Sollwert',
											eUnit				:= E_BA_Unit.eTime_Hours,
											fValue				:= 168);
											
	AblkFnct		: FB_AntBlkg; // Antiblockierschutzfunktion Pumpe	// anti-blocking protection function pump
END_VAR

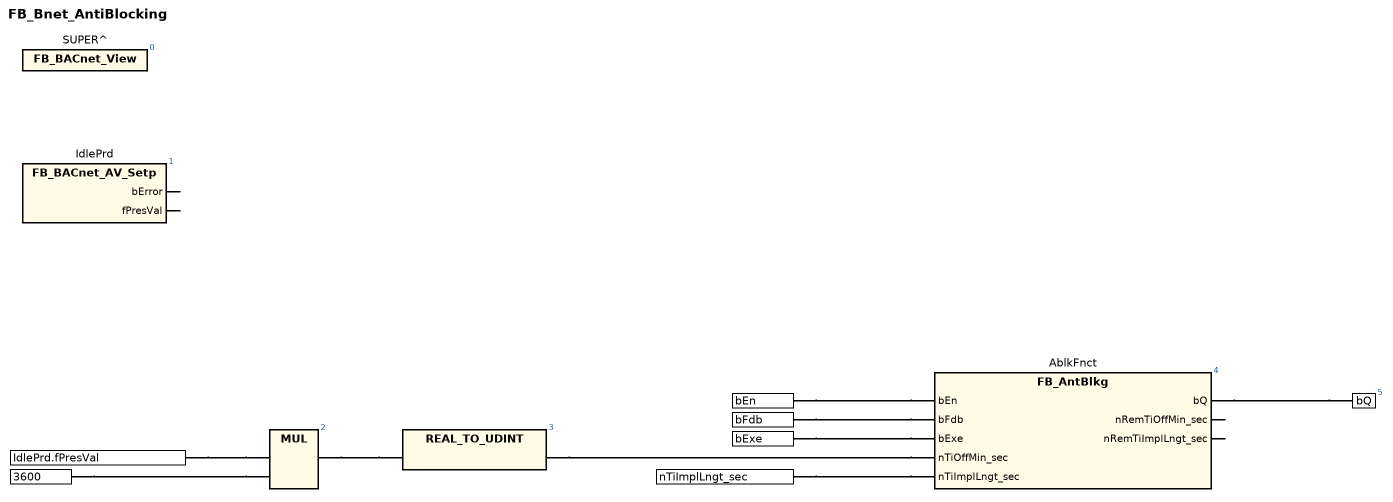
SUPER^(); // FB_BACnet_View
IdlePrd(); // FB_BACnet_AV_Setp
AblkFnct(
    bEn := bEn,
    bFdb := bFdb,
    bExe := bExe,
    nTiOffMin_sec := REAL_TO_UDINT(IdlePrd.fPresVal * 3600),
    nTiImplLngt_sec := nTiImplLngt_sec); // FB_AntBlkg
bQ := AblkFnct.bQ;

METHOD FB_init : BOOL
VAR_INPUT
	bInitRetains : BOOL; // if TRUE, the retain variables are initialized (warm start / cold start)
	bInCopyCode : BOOL;  // if TRUE, the instance afterwards gets moved into the copy code (online change)
END_VAR
sObjectName		:= '\/RZ01';
sDescription	:= '\/Blockierschutz';
END_METHOD

END_FUNCTION_BLOCK

// TEST/TestPackage/Templates/Universal/AntiBlocking/FB_AntBlkg
FUNCTION_BLOCK FB_AntBlkg
VAR_INPUT
	bEn					: BOOL;// enables the function block
	bFdb				: BOOL;// input for connecting the feedback signal of a motor or valve
	bExe				: BOOL;// rising edge forces a pulse output
	nTiOffMin_sec		: UDINT;// (0..Const.nTiSec) minimum switch-off time [s]: A pulse is issued once the time nTiOffMin has elapsed without movement of the unit
	nTiImplLngt_sec		: UDINT;// (0..Const.nTiSec) length of the blocking protection pulse [s] at bQ
END_VAR
VAR_OUTPUT
	bQ                  : BOOL;// pulse output
	nRemTiOffMin_sec    : UDINT;// remaining time [s] before the next pulse is issued in the absence of movement
	nRemTiImplLngt_sec  : UDINT;// remaining residual time [s] of the pulse at bQ
END_VAR
VAR
	tonTiOffMin			: TON;
	tTiOffMin			: TIME;
	tonImplLngt			: TON;
	tImplLngt			: TIME;
	nStep				: INT;
END_VAR

(*============================*)
tTiOffMin := TO_TIME(1000 * nTiOffMin_sec);
tImplLngt := TO_TIME(1000 * nTiImplLngt_sec);
(*============================*)

CASE nStep OF
0:
	nRemTiImplLngt_sec := 0;
	bQ := FALSE;
	tonImplLngt(IN := FALSE, PT := T#0s);
	tonTiOffMin(IN := bEn AND NOT bFdb, PT := tTiOffMin);
	nRemTiOffMin_sec := F_RemSecsTon(tonTimer := tonTiOffMin);

	IF	tonTiOffMin.Q AND bExe
	THEN
		bQ := TRUE;
		nStep := 10;
	END_IF

10:
	nRemTiOffMin_sec := 0;
	tonTiOffMin(IN := FALSE, PT := T#0s);
	tonImplLngt(IN := TRUE, PT := tImplLngt);
	nRemTiImplLngt_sec := F_RemSecsTon(tonTimer := tonImplLngt);

	IF	tonImplLngt.Q OR
		NOT bEn
	THEN
		nStep := 0;
	END_IF
END_CASE

END_FUNCTION_BLOCK

// TEST/TestPackage/Samples/Project Structure/PRG02/TEMPLATES/Custom/H/HtgCirABC123/FB_BA_HtgCirABC123_Vlv
FUNCTION_BLOCK FB_BA_HtgCirABC123_Vlv EXTENDS FB_BACnet_View
VAR_INPUT
	bEnSfty			: BOOL;
	fValSfty		: REAL;
	bEnCrit			: BOOL;
	fValCrit		: REAL;
	fValPgm			: REAL;
END_VAR
VAR_OUTPUT
	fPresentValue	: REAL;
	bEvent			: BOOL;
END_VAR
VAR
	AO								: FB_BACnet_AO_IO5P := (
										iParent 				:= THIS^,
										sObjectName				:= '\/CMD01',
										sDescription			:= '\/Schaltbefehl',
										sDeviceType				:= 'Ventil',
										fResolution				:= 0.003051851,
										fScaleOffset			:= 0,
										eUnit					:= E_BA_Unit.eOther_Percent);
END_VAR

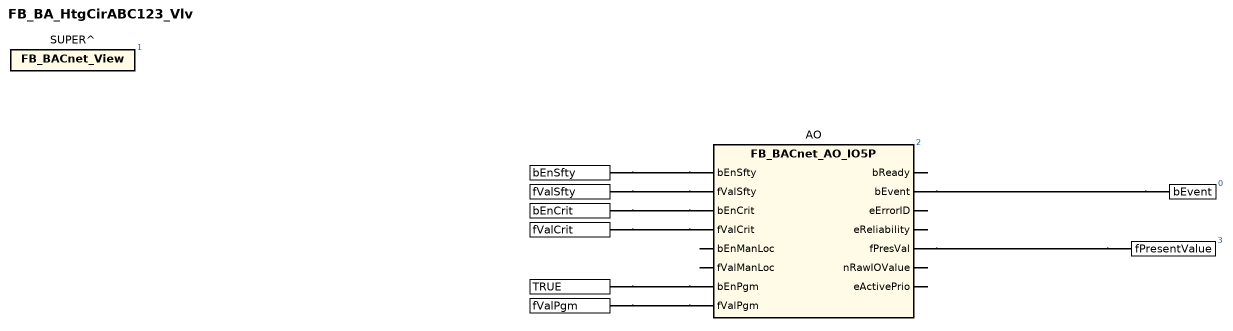
bEvent := AO.bEvent;
SUPER^(); // FB_BACnet_View
AO(
    bEnSfty := bEnSfty,
    fValSfty := fValSfty,
    bEnCrit := bEnCrit,
    fValCrit := fValCrit,
    bEnPgm := TRUE,
    fValPgm := fValPgm); // FB_BACnet_AO_IO5P
fPresentValue := AO.fPresVal;

METHOD FB_init : BOOL
VAR_INPUT
	bInitRetains : BOOL; // if TRUE, the retain variables are initialized (warm start / cold start)
	bInCopyCode : BOOL;  // if TRUE, the instance afterwards gets moved into the copy code (online change)
END_VAR
sObjectName		:= '\/VLV01';
sDescription	:= '\/Ventil';
END_METHOD

END_FUNCTION_BLOCK

// TEST/TestPackage/Samples/Project Structure/PRG02/TEMPLATES/Custom/H/HtgCirTZU555/FB_BA_HtgCirTZU555
FUNCTION_BLOCK FB_BA_HtgCirTZU555 EXTENDS FB_BACnet_View
VAR_INPUT CONSTANT
	WthT							: FB_BACnet_AI_IO := (
										iParent 					:= THIS^,
										sObjectName					:= '\/WTHT',
										sDescription				:= '\/Aussentemperatur',
										sDeviceType					:= 'Temperatursensor',
										fResolution					:= 0.003051851,
										eUnit						:= E_BA_Unit.eTemperature_DegreesCelsius);
										
	FlWT							: FB_BACnet_AI_IO := (
										iParent 					:= THIS^,
										sObjectName					:= '\/TVL',
										sDescription				:= '\/Vorlauftemperatur',
										sDeviceType					:= 'Temperatursensor',
										fResolution					:= 0.003051851,
										eUnit						:= E_BA_Unit.eTemperature_DegreesCelsius);
	RtWT							: FB_BACnet_AI_IO := (
										iParent 					:= THIS^,
										sObjectName					:= '\/TRT',
										sDescription				:= '\/Rücklauftemperatur',
										sDeviceType					:= 'Temperatursensor',
										fResolution					:= 0.003051851,
										fScaleOffset				:= 0,
										eUnit						:= E_BA_Unit.eTemperature_DegreesCelsius);
										
	Sched							: FB_BACnet_SchedB := (
										iParent 					:= THIS^,
										sObjectName					:= '\/SCH01',
										sDescription				:= '\/Zeitschaltprogramm',
										aWeek						:= F_BACnet_SchedWeekly3xB(E_BA_Weekday.eMonday, E_BA_Weekday.eFriday, T#0H, FALSE, T#6H, TRUE, T#20H, FALSE));
										
	PID								: FB_BACnet_Loop := (
										iParent 					:= THIS^,
										sObjectName					:= '\/PID01',
										sDescription				:= '\/Vorlauftemperatirregler',
										eAction						:= E_BA_Action.eReverse,
										fProportionalConstant		:= 1,
										fIntegralConstant			:= 180);	
										
	OpM								: FB_Bnet_H_OpM := (
										iParent 					:= THIS^);	
										
	SpG								: FB_Bnet_H_HtgCir_Sp := (
										iParent 					:= THIS^);	
										
	HtgLimit						: FB_Bnet_H_HtgCir_HtgLmt := (
										iParent 					:= THIS^);
										
	Vlv								: FB_Bnet_Vlv_013 := (
										iParent 					:= THIS^);	
										
	Pu								: FB_Bnet_Pu1st := (
										iParent 					:= THIS^);	
END_VAR
VAR // added by the converter: edge detectors and wires of the graphical bodies
    _w1 : ANY;
END_VAR

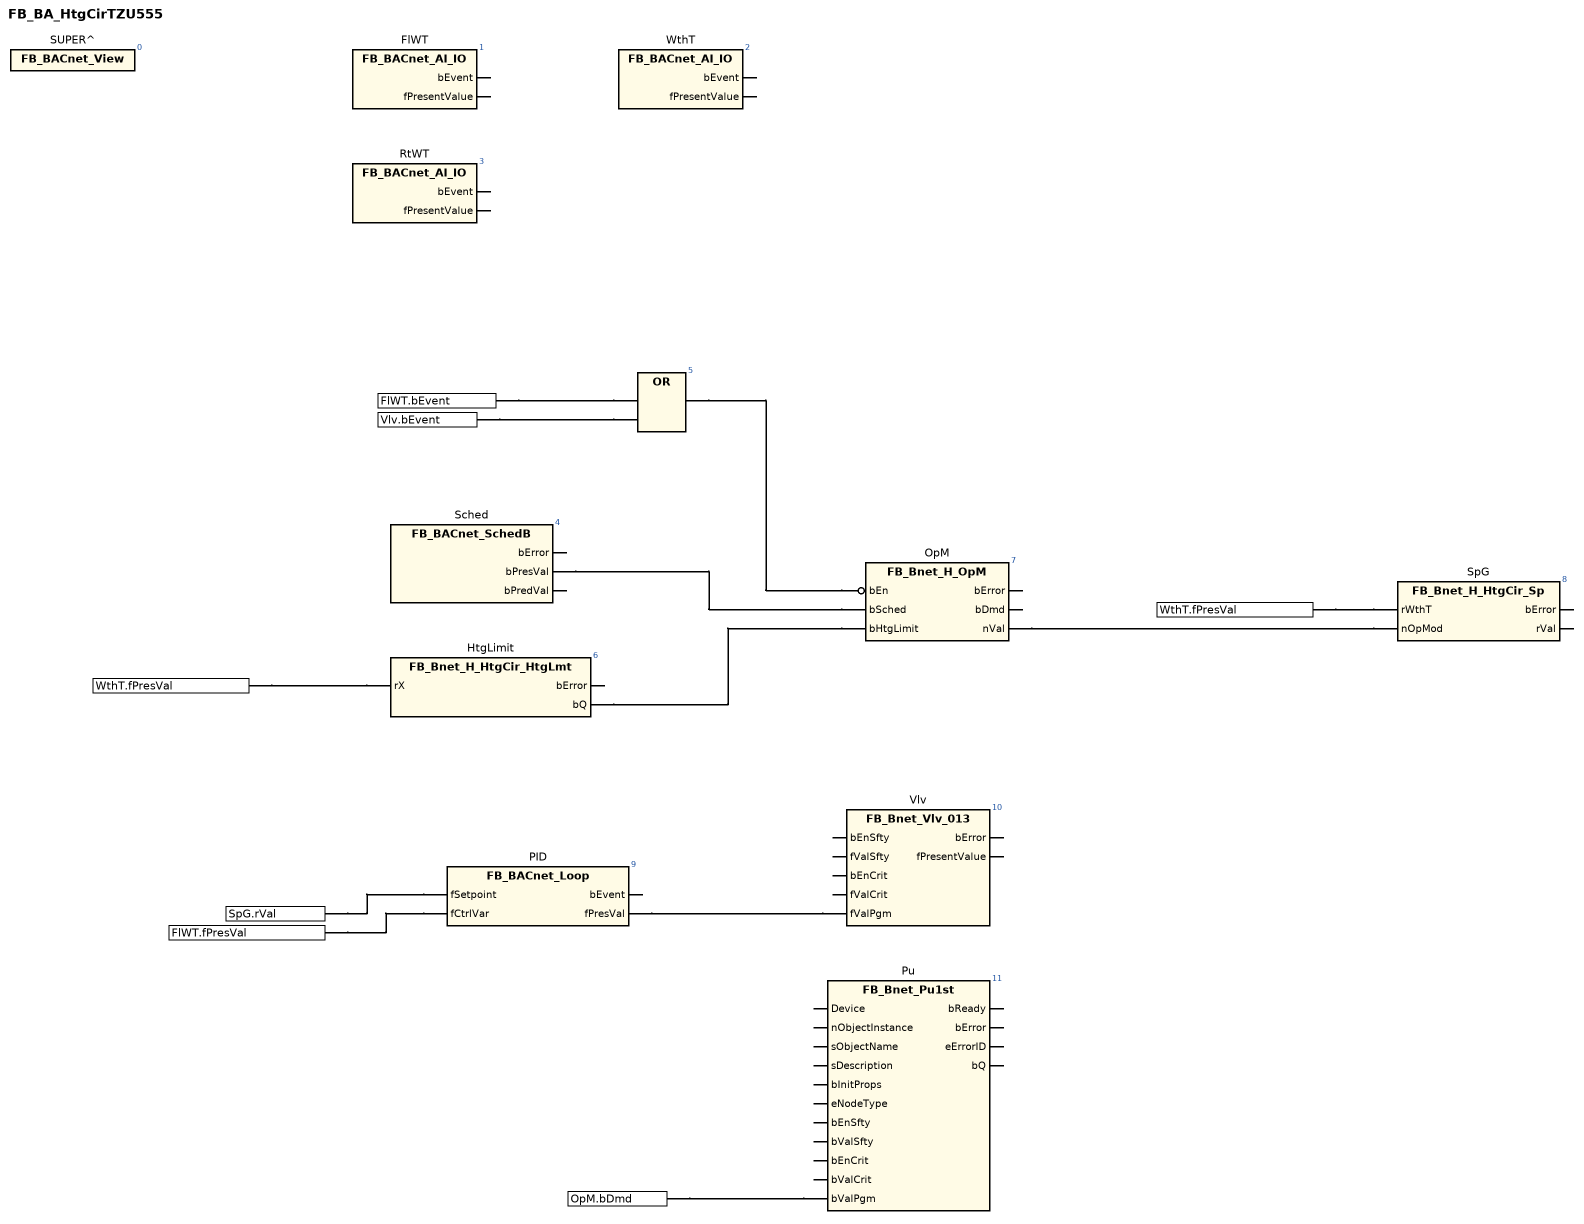
// note: 28 stored wires end on pins the file does not list and are not shown
SUPER^(); // FB_BACnet_View
FlWT(); // FB_BACnet_AI_IO
WthT(); // FB_BACnet_AI_IO
RtWT(); // FB_BACnet_AI_IO
Sched(); // FB_BACnet_SchedB
_w1 := FlWT.bEvent OR Vlv.bEvent;
HtgLimit(rX := WthT.fPresVal); // FB_Bnet_H_HtgCir_HtgLmt
OpM(bEn := NOT _w1, bSched := Sched.bPresVal, bHtgLimit := HtgLimit.bQ); // FB_Bnet_H_OpM
SpG(rWthT := WthT.fPresVal, nOpMod := OpM.nVal); // FB_Bnet_H_HtgCir_Sp
PID(fSetpoint := SpG.rVal, fCtrlVar := FlWT.fPresVal); // FB_BACnet_Loop
Vlv(fValPgm := PID.fPresVal); // FB_Bnet_Vlv_013
Pu(bValPgm := OpM.bDmd); // FB_Bnet_Pu1st

METHOD FB_init : BOOL
VAR_INPUT
	bInitRetains : BOOL; // if TRUE, the retain variables are initialized (warm start / cold start)
	bInCopyCode : BOOL;  // if TRUE, the instance afterwards gets moved into the copy code (online change)
END_VAR
sObjectName		:= '\/HCR01';
sDescription	:= '\/Heizkreis';

Pu.BO.sObjectName := '\/XXXtest';
END_METHOD

END_FUNCTION_BLOCK

// TEST/TestPackage/Samples/Project Structure/PRG02/TEMPLATES/Custom/H/HtgCirTZU555/FB_BA_HtgCirTZU555_Pu
FUNCTION_BLOCK FB_BA_HtgCirTZU555_Pu EXTENDS FB_BACnet_View
VAR_INPUT
	bEnSfty			: BOOL;
	fValSfty		: REAL;
	bEnCrit			: BOOL;
	fValCrit		: REAL;
	fValPgm			: REAL;
END_VAR
VAR_OUTPUT
	fPresentValue	: REAL;
	bEvent			: BOOL;
END_VAR
VAR
	AO								: FB_BACnet_AO_IO5P := (
										iParent 				:= THIS^,
										sObjectName				:= '\/CMD01',
										sDescription			:= '\/Schaltbefehl',
										sDeviceType				:= 'Ventil',
										fResolution				:= 0.003051851,
										fScaleOffset			:= 0,
										eUnit					:= E_BA_Unit.eOther_Percent);
END_VAR

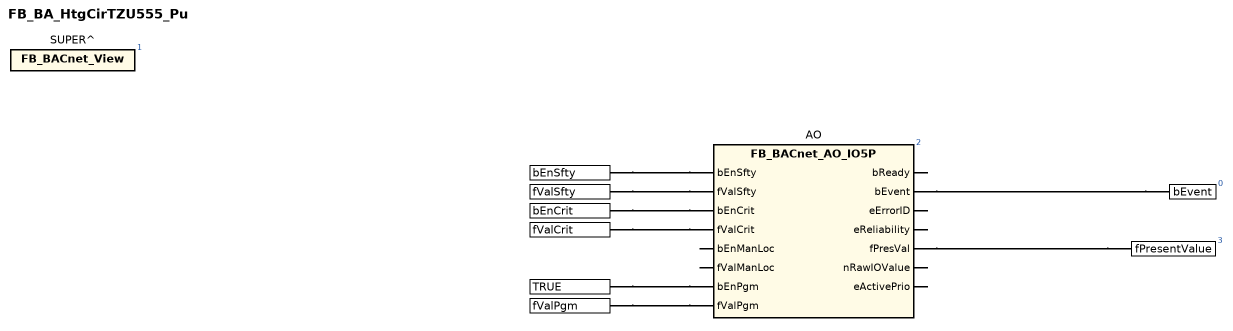
bEvent := AO.bEvent;
SUPER^(); // FB_BACnet_View
AO(
    bEnSfty := bEnSfty,
    fValSfty := fValSfty,
    bEnCrit := bEnCrit,
    fValCrit := fValCrit,
    bEnPgm := TRUE,
    fValPgm := fValPgm); // FB_BACnet_AO_IO5P
fPresentValue := AO.fPresVal;

METHOD FB_init : BOOL
VAR_INPUT
	bInitRetains : BOOL; // if TRUE, the retain variables are initialized (warm start / cold start)
	bInCopyCode : BOOL;  // if TRUE, the instance afterwards gets moved into the copy code (online change)
END_VAR
sObjectName		:= '\/VLV01';
sDescription	:= '\/Ventil';
END_METHOD

END_FUNCTION_BLOCK

// TEST/TestPackage/Samples/Project Structure/PRG02/TEMPLATES/Standard/AC/FB_BACnet_AC01
FUNCTION_BLOCK FB_BACnet_AC01 EXTENDS FB_BACnet_View
VAR_INPUT CONSTANT
	WthT							: FB_BACnet_AI_IO := (
										iParent 					:= THIS^,
										sObjectName					:= '\/WTHT',
										sDescription				:= '\/Aussentemperatur',
										sDeviceType					:= 'Temperatursensor',
										fResolution					:= 0.003051851,
										eUnit						:= E_BA_Unit.eTemperature_DegreesCelsius);
										
	FlWT							: FB_BACnet_AI_IO := (
										iParent 					:= THIS^,
										sObjectName					:= '\/TVL',
										sDescription				:= '\/Vorlauftemperatur',
										sDeviceType					:= 'Temperatursensor',
										fResolution					:= 0.003051851,
										eUnit						:= E_BA_Unit.eTemperature_DegreesCelsius);
	RtWT							: FB_BACnet_AI_IO := (
										iParent 					:= THIS^,
										sObjectName					:= '\/TRT',
										sDescription				:= '\/Rücklauftemperatur',
										sDeviceType					:= 'Temperatursensor',
										fResolution					:= 0.003051851,
										fScaleOffset				:= 0,
										eUnit						:= E_BA_Unit.eTemperature_DegreesCelsius);
										
	Sched							: FB_BACnet_SchedB := (
										iParent 					:= THIS^,
										sObjectName					:= '\/SCH01',
										sDescription				:= '\/Zeitschaltprogramm',
										aWeek						:= F_BACnet_SchedWeekly3xB(E_BA_Weekday.eMonday, E_BA_Weekday.eFriday, T#0H, FALSE, T#6H, TRUE, T#20H, FALSE));
										
	PID								: FB_BACnet_Loop := (
										iParent 					:= THIS^,
										sObjectName					:= '\/PID01',
										sDescription				:= '\/Vorlauftemperatirregler',
										eAction						:= E_BA_Action.eReverse,
										fProportionalConstant		:= 1,
										fIntegralConstant			:= 180);	
										
	OpM								: FB_Bnet_H_OpM := (
										iParent 					:= THIS^);	
										
	SpG								: FB_Bnet_H_HtgCir_Sp := (
										iParent 					:= THIS^);	
										
	HtgLimit						: FB_Bnet_H_HtgCir_HtgLmt := (
										iParent 					:= THIS^);
										
	Vlv								: FB_Bnet_Vlv_013 := (
										iParent 					:= THIS^);	
										
	Pu								: FB_Bnet_Pu1st := (
										iParent 					:= THIS^);	
END_VAR
VAR // added by the converter: edge detectors and wires of the graphical bodies
    _w1 : ANY;
END_VAR

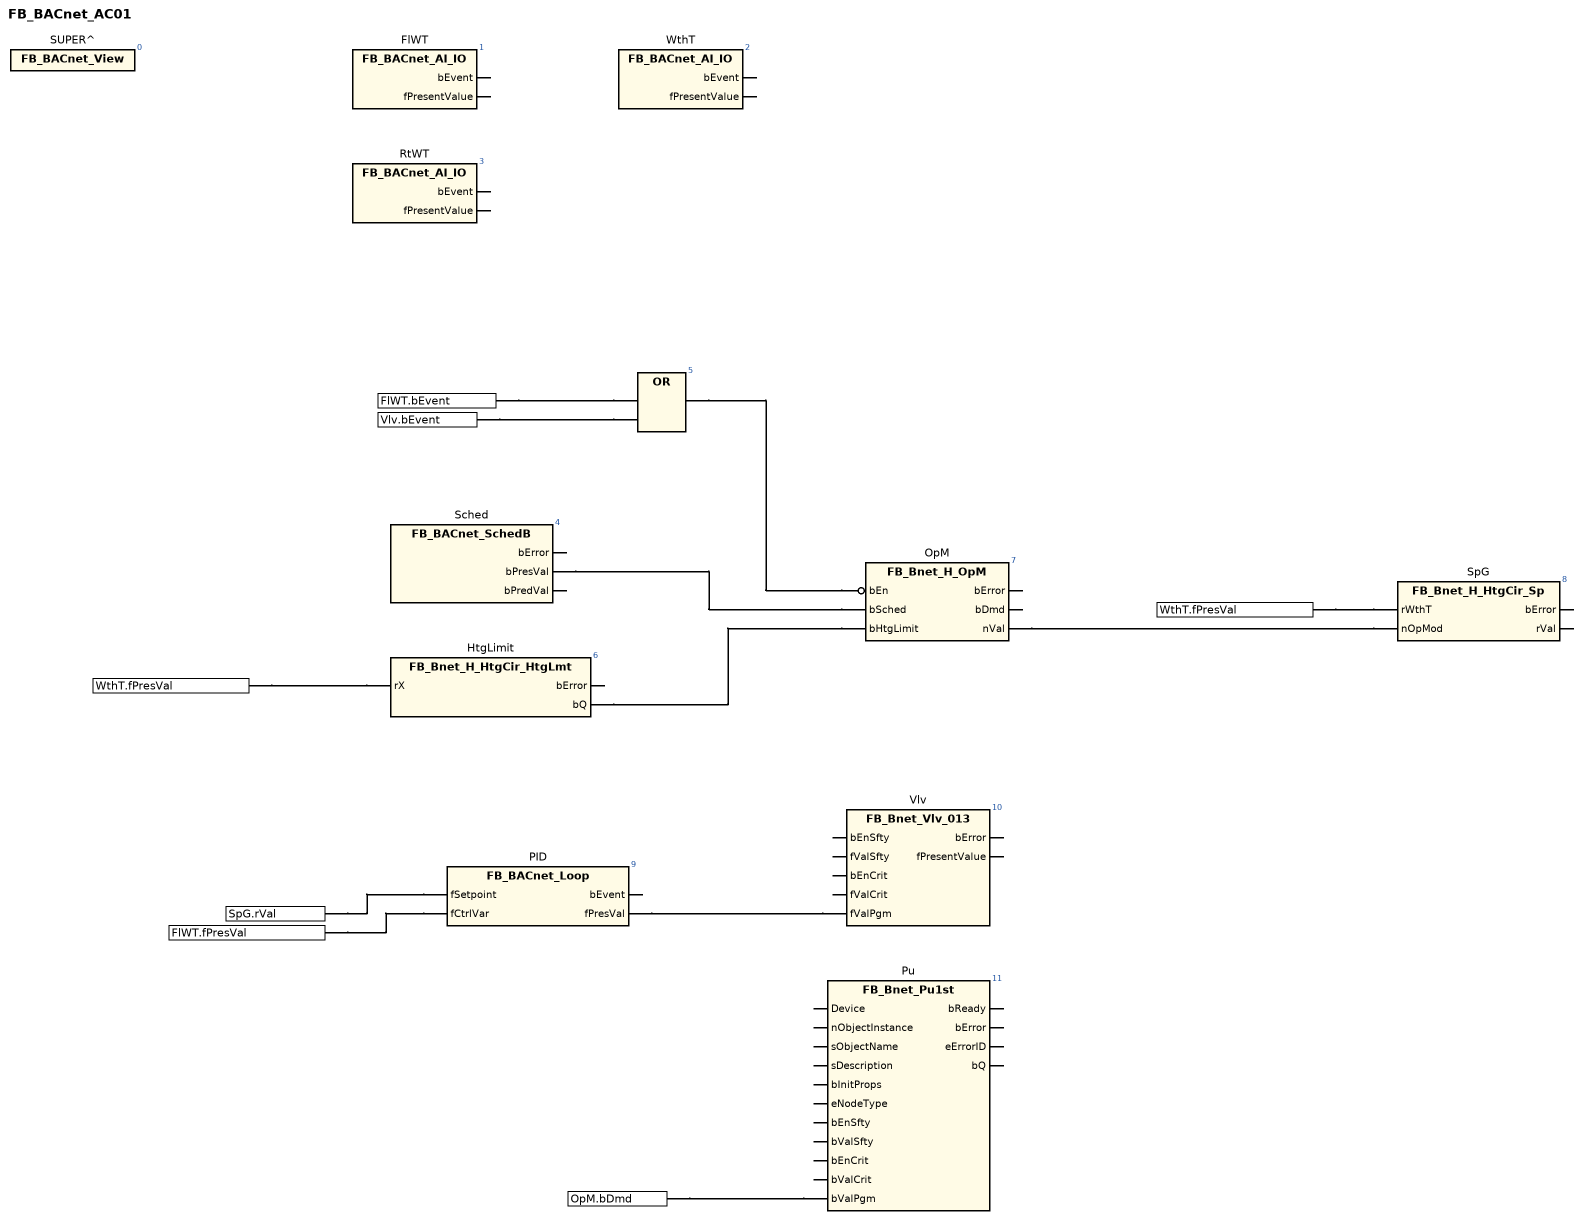
// note: 28 stored wires end on pins the file does not list and are not shown
SUPER^(); // FB_BACnet_View
FlWT(); // FB_BACnet_AI_IO
WthT(); // FB_BACnet_AI_IO
RtWT(); // FB_BACnet_AI_IO
Sched(); // FB_BACnet_SchedB
_w1 := FlWT.bEvent OR Vlv.bEvent;
HtgLimit(rX := WthT.fPresVal); // FB_Bnet_H_HtgCir_HtgLmt
OpM(bEn := NOT _w1, bSched := Sched.bPresVal, bHtgLimit := HtgLimit.bQ); // FB_Bnet_H_OpM
SpG(rWthT := WthT.fPresVal, nOpMod := OpM.nVal); // FB_Bnet_H_HtgCir_Sp
PID(fSetpoint := SpG.rVal, fCtrlVar := FlWT.fPresVal); // FB_BACnet_Loop
Vlv(fValPgm := PID.fPresVal); // FB_Bnet_Vlv_013
Pu(bValPgm := OpM.bDmd); // FB_Bnet_Pu1st

METHOD FB_init : BOOL
VAR_INPUT
	bInitRetains : BOOL; // if TRUE, the retain variables are initialized (warm start / cold start)
	bInCopyCode : BOOL;  // if TRUE, the instance afterwards gets moved into the copy code (online change)
END_VAR
sObjectName		:= '\/HCR01';
sDescription	:= '\/Heizkreis';

Pu.BO.sObjectName := '\/XXXtest';
END_METHOD

END_FUNCTION_BLOCK

// TEST/TestPackage/Samples/Project Structure/PRG02/TEMPLATES/Standard/H/FB_BACnet_HtgCir01
FUNCTION_BLOCK FB_BACnet_HtgCir01 EXTENDS FB_BACnet_View
VAR_INPUT CONSTANT
	WthT							: FB_BACnet_AI_IO := (
										iParent 					:= THIS^,
										sObjectName					:= '\/WTHT',
										sDescription				:= '\/Aussentemperatur',
										sDeviceType					:= 'Temperatursensor',
										fResolution					:= 0.003051851,
										eUnit						:= E_BA_Unit.eTemperature_DegreesCelsius);
										
	FlWT							: FB_BACnet_AI_IO := (
										iParent 					:= THIS^,
										sObjectName					:= '\/TVL',
										sDescription				:= '\/Vorlauftemperatur',
										sDeviceType					:= 'Temperatursensor',
										fResolution					:= 0.003051851,
										eUnit						:= E_BA_Unit.eTemperature_DegreesCelsius);
	RtWT							: FB_BACnet_AI_IO := (
										iParent 					:= THIS^,
										sObjectName					:= '\/TRT',
										sDescription				:= '\/Rücklauftemperatur',
										sDeviceType					:= 'Temperatursensor',
										fResolution					:= 0.003051851,
										fScaleOffset				:= 0,
										eUnit						:= E_BA_Unit.eTemperature_DegreesCelsius);
										
	Sched							: FB_BACnet_SchedB := (
										iParent 					:= THIS^,
										sObjectName					:= '\/SCH01',
										sDescription				:= '\/Zeitschaltprogramm',
										aWeek						:= F_BACnet_SchedWeekly3xB(E_BA_Weekday.eMonday, E_BA_Weekday.eFriday, T#0H, FALSE, T#6H, TRUE, T#20H, FALSE));
										
	PID								: FB_BACnet_Loop := (
										iParent 					:= THIS^,
										sObjectName					:= '\/PID01',
										sDescription				:= '\/Vorlauftemperatirregler',
										eAction						:= E_BA_Action.eReverse,
										fProportionalConstant		:= 1,
										fIntegralConstant			:= 180);	
										
	OpM								: FB_Bnet_H_OpM := (
										iParent 					:= THIS^);	
										
	SpG								: FB_Bnet_H_HtgCir_Sp := (
										iParent 					:= THIS^);	
										
	HtgLimit						: FB_Bnet_H_HtgCir_HtgLmt := (
										iParent 					:= THIS^);
										
	Vlv								: FB_Bnet_Vlv_013 := (
										iParent 					:= THIS^);	
										
	Pu								: FB_Bnet_Pu1st := (
										iParent 					:= THIS^);	
END_VAR
VAR // added by the converter: edge detectors and wires of the graphical bodies
    _w1 : ANY;
END_VAR

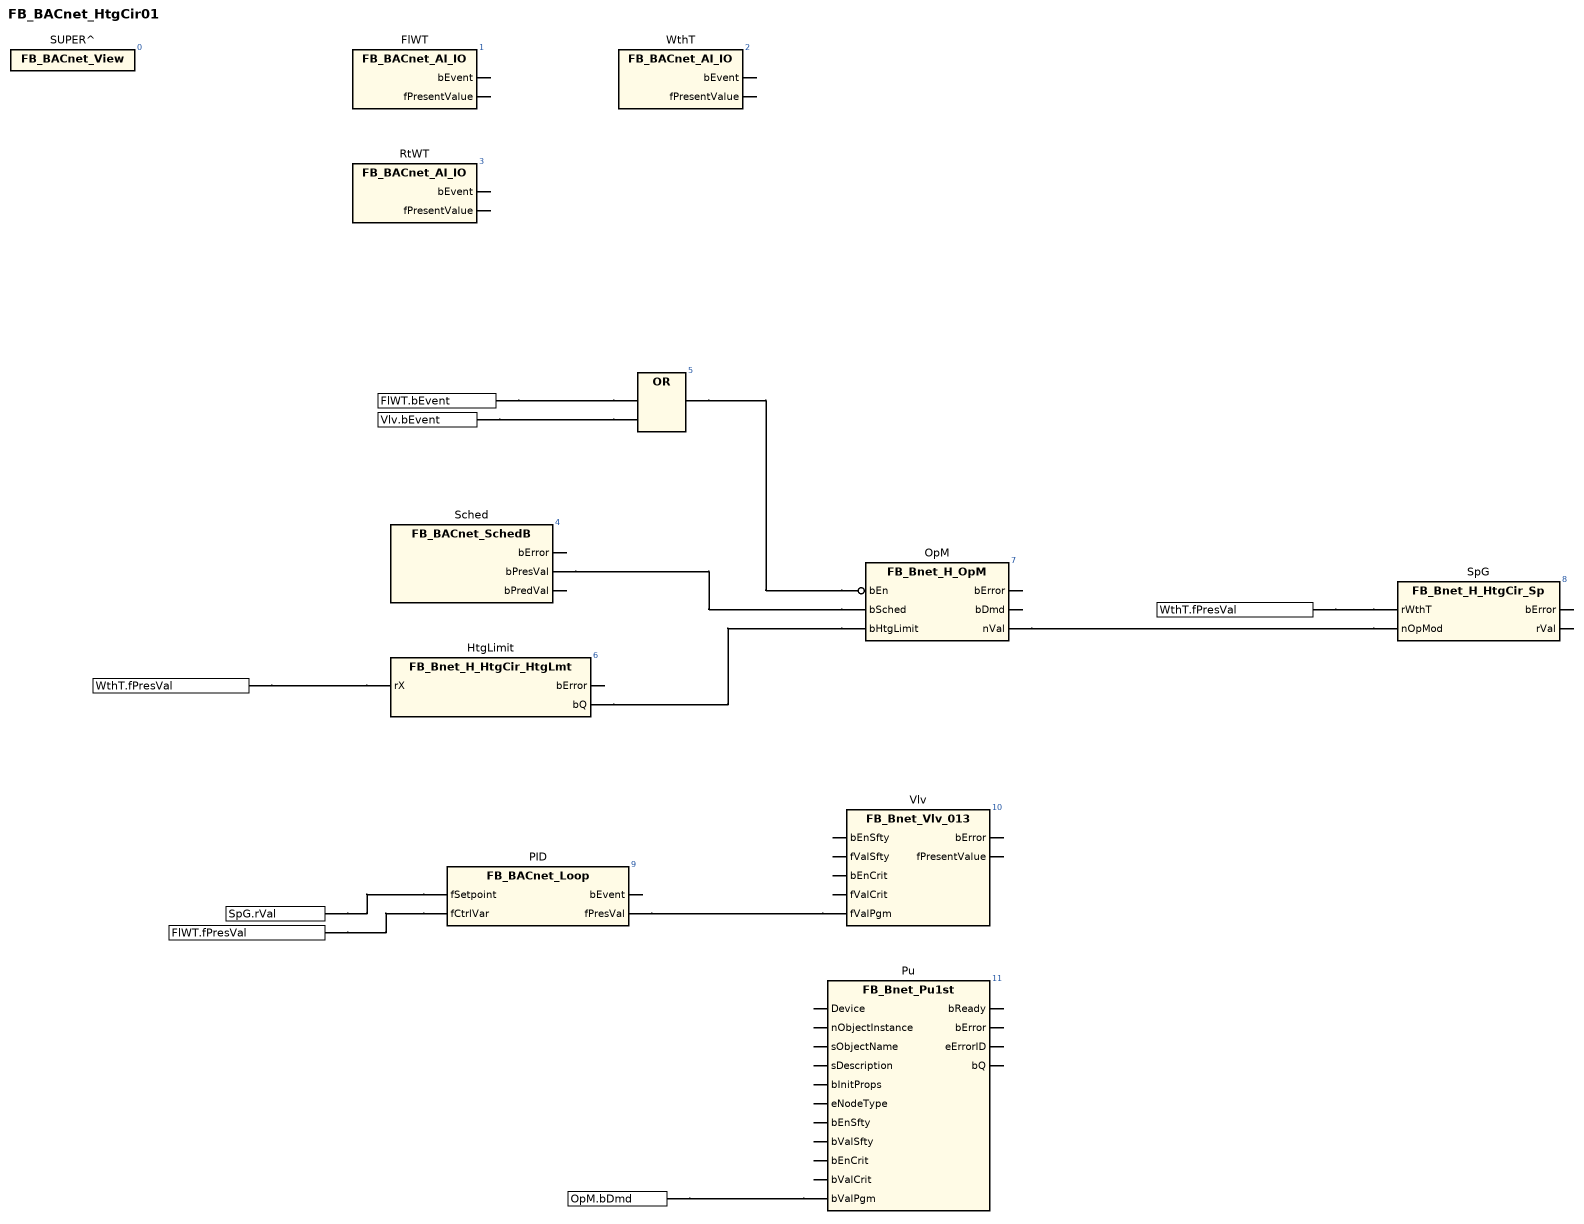
// note: 28 stored wires end on pins the file does not list and are not shown
SUPER^(); // FB_BACnet_View
FlWT(); // FB_BACnet_AI_IO
WthT(); // FB_BACnet_AI_IO
RtWT(); // FB_BACnet_AI_IO
Sched(); // FB_BACnet_SchedB
_w1 := FlWT.bEvent OR Vlv.bEvent;
HtgLimit(rX := WthT.fPresVal); // FB_Bnet_H_HtgCir_HtgLmt
OpM(bEn := NOT _w1, bSched := Sched.bPresVal, bHtgLimit := HtgLimit.bQ); // FB_Bnet_H_OpM
SpG(rWthT := WthT.fPresVal, nOpMod := OpM.nVal); // FB_Bnet_H_HtgCir_Sp
PID(fSetpoint := SpG.rVal, fCtrlVar := FlWT.fPresVal); // FB_BACnet_Loop
Vlv(fValPgm := PID.fPresVal); // FB_Bnet_Vlv_013
Pu(bValPgm := OpM.bDmd); // FB_Bnet_Pu1st

METHOD FB_init : BOOL
VAR_INPUT
	bInitRetains : BOOL; // if TRUE, the retain variables are initialized (warm start / cold start)
	bInCopyCode : BOOL;  // if TRUE, the instance afterwards gets moved into the copy code (online change)
END_VAR
sObjectName		:= '\/HCR01';
sDescription	:= '\/Heizkreis';

Pu.BO.sObjectName := '\/XXXtest';
END_METHOD

END_FUNCTION_BLOCK

// TEST/TestPackage/Samples/Project Structure/PRG02/TEMPLATES/Standard/Universal/Valve/FB_Bnet_Vlv_014
FUNCTION_BLOCK FB_Bnet_Vlv_014 EXTENDS FB_BACnet_View
VAR_INPUT
	bEnSfty			: BOOL;
	fValSfty		: REAL;
	bEnCrit			: BOOL;
	fValCrit		: REAL;
	fValPgm			: REAL;
END_VAR
VAR_OUTPUT
	fPresentValue	: REAL;
	bEvent			: BOOL;
END_VAR
VAR
	AO								: FB_BACnet_AO_IO5P := (
										iParent 				:= THIS^,
										sObjectName				:= '\/CMD01',
										sDescription			:= '\/Schaltbefehl',
										sDeviceType				:= 'Ventil',
										fResolution				:= 0.003051851,
										fScaleOffset			:= 0,
										eUnit					:= E_BA_Unit.eOther_Percent);
END_VAR

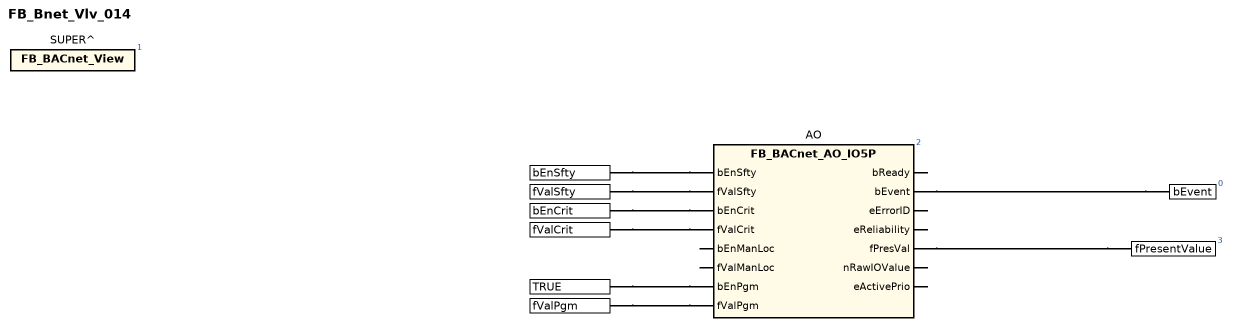
bEvent := AO.bEvent;
SUPER^(); // FB_BACnet_View
AO(
    bEnSfty := bEnSfty,
    fValSfty := fValSfty,
    bEnCrit := bEnCrit,
    fValCrit := fValCrit,
    bEnPgm := TRUE,
    fValPgm := fValPgm); // FB_BACnet_AO_IO5P
fPresentValue := AO.fPresVal;

METHOD FB_init : BOOL
VAR_INPUT
	bInitRetains : BOOL; // if TRUE, the retain variables are initialized (warm start / cold start)
	bInCopyCode : BOOL;  // if TRUE, the instance afterwards gets moved into the copy code (online change)
END_VAR
sObjectName		:= '\/VLV01';
sDescription	:= '\/Ventil';
END_METHOD

END_FUNCTION_BLOCK

// TEST/TestPackage/Samples/Project Structure/PRG02/MAIN_PRG02
PROGRAM MAIN_PRG02
VAR
	B01								: FB_BACnet_View		:= (						sObjectName := '\/B01',			sDescription := 'Gebäude 1');
		ISP01						: FB_BACnet_View		:= (iParent	:= B01,			sObjectName := '\/ISP01',		sDescription := 'Informationsschwerpunkt 1');
			H						: FB_BACnet_View		:= (iParent	:= ISP01,		sObjectName := '\/H',			sDescription := 'Heizungsanlagen');
				HtgCir01			: FB_BACnet_HtgCir01	:= (iParent	:= H,			sObjectName := '\/HTG01',		sDescription := 'Statischer Heizkreis 1');			// Hier ein Standard-Heizkreis
				HtgCir02			: FB_BACnet_HtgCir01	:= (iParent	:= H,			sObjectName := '\/HTG02',		sDescription := 'Statischer Heizkreis 2');			// Hier ein Standard-Heizkreis
				HtgCir03			: FB_BACnet_HtgCir01	:= (iParent	:= H,			sObjectName := '\/HTG03',		sDescription := 'Statischer Heizkreis 3');			// Hier ein Standard-Heizkreis
				HtgCirABC123		: FB_BA_HtgCirABC123	:= (iParent	:= H,			sObjectName := '\/HTG11',		sDescription := 'Heizkreis Kantine');				// Hier ein angepasster Heizkreis
				HtgCirTZU555		: FB_BA_HtgCirTZU555	:= (iParent	:= H,			sObjectName := '\/HTG12',		sDescription := 'Heizkreis Hausmeister');			// Hier ein angepasster Heizkreis + individualisierung
			AC						: FB_BACnet_View		:= (iParent	:= ISP01,		sObjectName := '\/AC',			sDescription := 'Lüftungsanlagen');
				AC01				: FB_BACnet_AC01		:= (iParent	:= AC,			sObjectName := '\/APLT01',		sDescription := 'Lüftungsanlage 1');				// Hier eine Standard-Lüftung
				AC02				: FB_BACnet_AC01		:= (iParent	:= AC,			sObjectName := '\/APLT02',		sDescription := 'Lüftungsanlage 2');				// Hier eine Standard-Lüftung
				AC03				: FB_BACnet_AC01		:= (iParent	:= AC,			sObjectName := '\/APLT03',		sDescription := 'Lüftungsanlage 3');				// Hier eine Standard-Lüftung
				AC04				: FB_BACnet_AC01		:= (iParent	:= AC,			sObjectName := '\/APLT04',		sDescription := 'Lüftungsanlage 4');				// Hier eine Standard-Lüftung
				AC05				: FB_BACnet_AC01		:= (iParent	:= AC,			sObjectName := '\/APLT05',		sDescription := 'Lüftungsanlage 5');				// Hier eine Standard-Lüftung
END_VAR

B01();
ISP01();
H();
HtgCir01();
HtgCir02();
HtgCir03();
HtgCirABC123();
HtgCirTZU555();
AC();
AC01();
AC02();
AC03();
AC04();
AC05();

END_PROGRAM

// TEST/TestPackage/Templates/HeatSupply/HeatingCircuit/Plants/FB_Bnet_H_HtgCir_01
FUNCTION_BLOCK FB_Bnet_H_HtgCir_01 EXTENDS FB_BACnet_View
VAR_INPUT CONSTANT
	WthT							: FB_BACnet_AI_IO := (
										iParent 					:= THIS^,
										sObjectName					:= '\/WTHT',
										sDescription				:= '\/Aussentemperatur',
										sDeviceType					:= 'Temperatursensor',
										fResolution					:= 0.003051851,
										eUnit						:= E_BA_Unit.eTemperature_DegreesCelsius);
										
	FlWT							: FB_BACnet_AI_IO := (
										iParent 					:= THIS^,
										sObjectName					:= '\/TVL',
										sDescription				:= '\/Vorlauftemperatur',
										sDeviceType					:= 'Temperatursensor',
										fResolution					:= 0.003051851,
										eUnit						:= E_BA_Unit.eTemperature_DegreesCelsius);
	RtWT							: FB_BACnet_AI_IO := (
										iParent 					:= THIS^,
										sObjectName					:= '\/TRT',
										sDescription				:= '\/Rücklauftemperatur',
										sDeviceType					:= 'Temperatursensor',
										fResolution					:= 0.003051851,
										fScaleOffset				:= 0,
										eUnit						:= E_BA_Unit.eTemperature_DegreesCelsius);
										
	Sched							: FB_BACnet_SchedB := (
										iParent 					:= THIS^,
										sObjectName					:= '\/SCH01',
										sDescription				:= '\/Zeitschaltprogramm',
										aWeek						:= F_BACnet_SchedWeekly3xB(E_BA_Weekday.eMonday, E_BA_Weekday.eFriday, T#0H, FALSE, T#6H, TRUE, T#20H, FALSE));
										
	PID								: FB_BACnet_Loop := (
										iParent 					:= THIS^,
										sObjectName					:= '\/PID01',
										sDescription				:= '\/Vorlauftemperaturregler',
										eAction						:= E_BA_Action.eReverse,
										fProportionalConstant		:= 1,
										fIntegralConstant			:= 180);	
										
	OpM								: FB_Bnet_H_OpM := (
										iParent 					:= THIS^);	
										
	SpG								: FB_Bnet_H_HtgCir_Sp := (
										iParent 					:= THIS^);	
										
	HtgLimit						: FB_Bnet_H_HtgCir_HtgLmt := (
										iParent 					:= THIS^);
										
	Vlv								: FB_Bnet_Vlv_013 := (
										iParent 					:= THIS^);	
										
	Pu								: FB_Bnet_Pu1st := (
										iParent 					:= THIS^);	
END_VAR
VAR // added by the converter: edge detectors and wires of the graphical bodies
    _w1 : ANY;
END_VAR

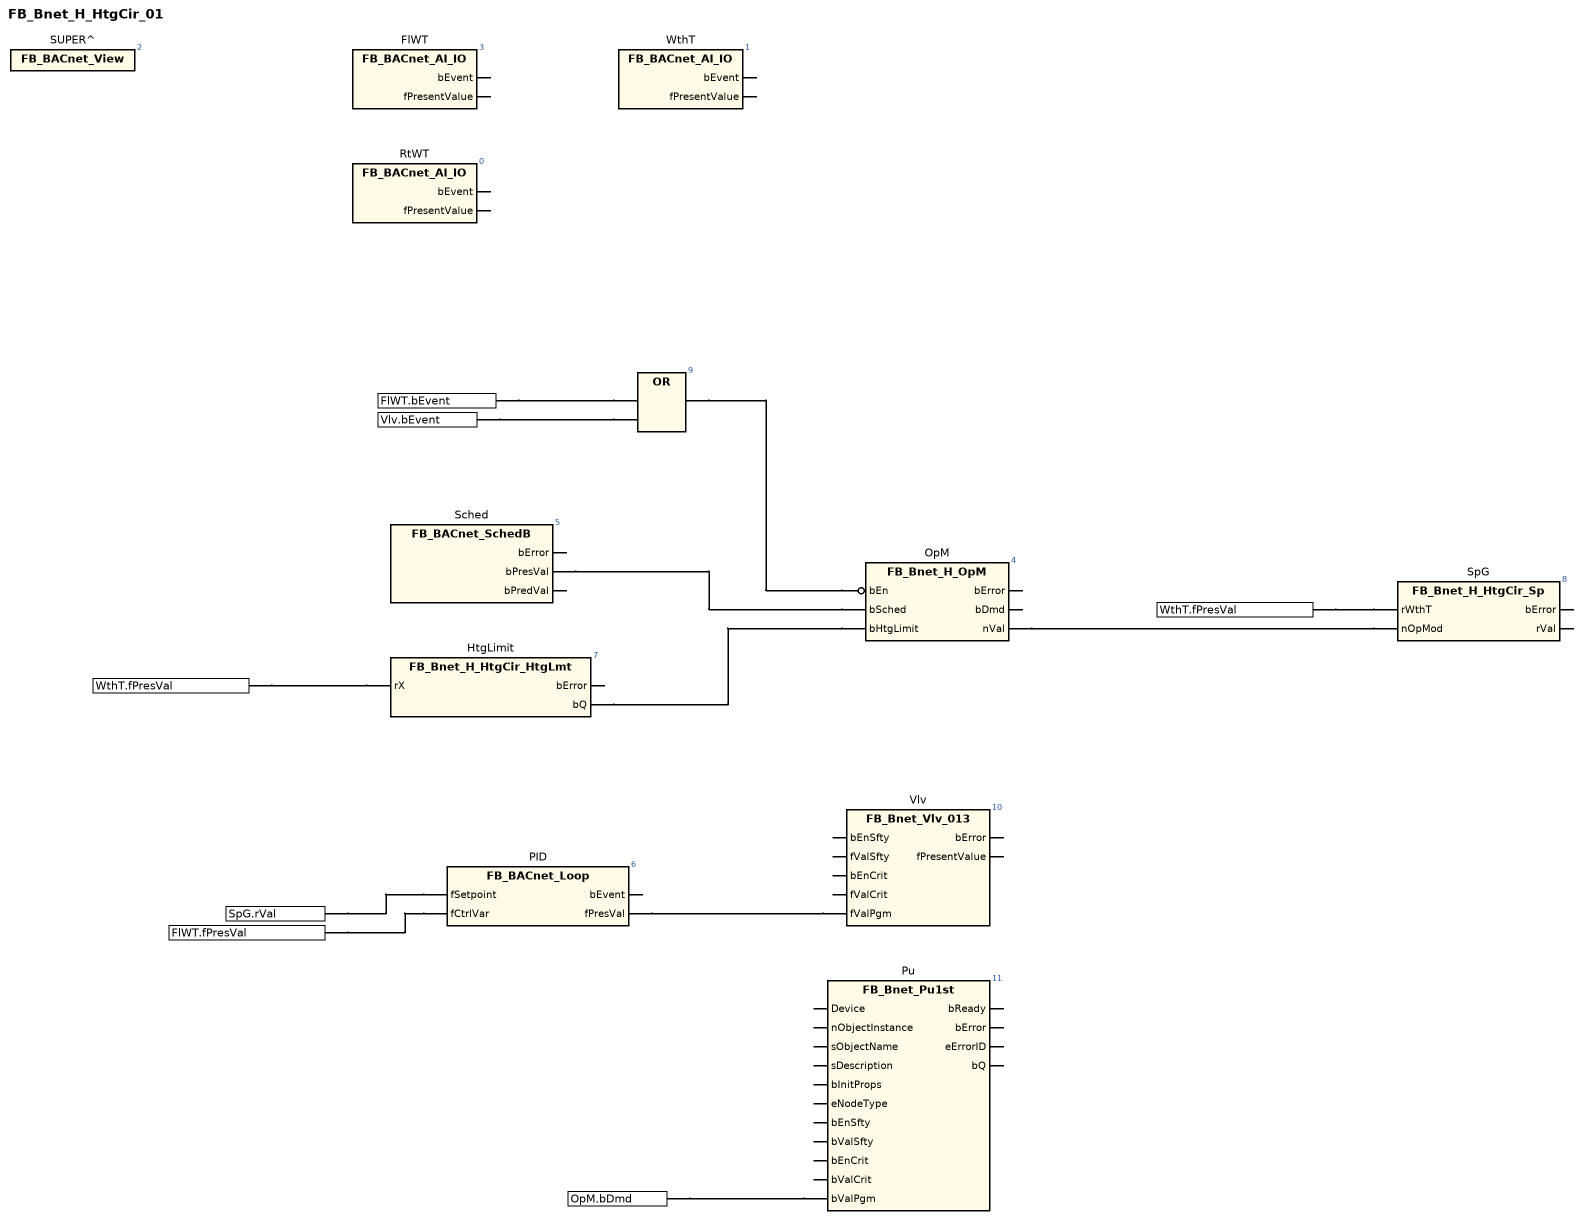
// note: 28 stored wires end on pins the file does not list and are not shown
RtWT(); // FB_BACnet_AI_IO
WthT(); // FB_BACnet_AI_IO
SUPER^(); // FB_BACnet_View
FlWT(); // FB_BACnet_AI_IO
OpM(bEn := NOT _w1, bSched := Sched.bPresVal, bHtgLimit := HtgLimit.bQ); // FB_Bnet_H_OpM
Sched(); // FB_BACnet_SchedB
PID(fSetpoint := SpG.rVal, fCtrlVar := FlWT.fPresVal); // FB_BACnet_Loop
HtgLimit(rX := WthT.fPresVal); // FB_Bnet_H_HtgCir_HtgLmt
SpG(rWthT := WthT.fPresVal, nOpMod := OpM.nVal); // FB_Bnet_H_HtgCir_Sp
_w1 := FlWT.bEvent OR Vlv.bEvent;
Vlv(fValPgm := PID.fPresVal); // FB_Bnet_Vlv_013
Pu(bValPgm := OpM.bDmd); // FB_Bnet_Pu1st

METHOD FB_init : BOOL
VAR_INPUT
	bInitRetains : BOOL; // if TRUE, the retain variables are initialized (warm start / cold start)
	bInCopyCode : BOOL;  // if TRUE, the instance afterwards gets moved into the copy code (online change)
END_VAR
sObjectName		:= '\/HCR01';
sDescription	:= '\/Heizkreis';

Pu.BO.sObjectName := '\/XXXtest';
END_METHOD

END_FUNCTION_BLOCK

